LIN {X 0,Y 631.994,Z 1164.814,A -85,B 0,C 180,E1 28881.357,E2 28881.357} C_VEL
LIN {X 0,Y 632.102,Z 1158.024,A -85,B 0,C 180,E1 28878.874,E2 28878.874} C_VEL
LIN {X 0,Y 632.325,Z 1150.394,A -85,B 0,C 180,E1 28876.653,E2 28876.653} C_VEL
LIN {X 0,Y 632.601,Z 1142.497,A -85,B 0,C 180,E1 28874.696,E2 28874.696} C_VEL
LIN {X 0,Y 633.008,Z 1133.821,A -85,B 0,C 180,E1 28872.821,E2 28872.821} C_VEL
LIN {X 0,Y 633.525,Z 1124.191,A -85,B 0,C 180,E1 28870.98,E2 28870.98} C_VEL
LIN {X 0,Y 634.156,Z 1113.94,A -85,B 0,C 180,E1 28869.223,E2 28869.223} C_VEL
LIN {X 0,Y 635.003,Z 1101.645,A -85,B 0,C 180,E1 28867.329,E2 28867.329} C_VEL
LIN {X 0,Y 636.328,Z 1084.564,A -85,B 0,C 180,E1 28864.997,E2 28864.997} C_VEL
LIN {X 0,Y 637.814,Z 1067.276,A -85,B 0,C 180,E1 28862.93,E2 28862.93} C_VEL
LIN {X 0,Y 639.378,Z 1049.829,A -85,B 0,C 180,E1 28861.064,E2 28861.064} C_VEL
LIN {X 0,Y 641.404,Z 1029.08,A -85,B 0,C 180,E1 28859.094,E2 28859.094} C_VEL
LIN {X 0,Y 643.497,Z 1007.241,A -85,B 0,C 180,E1 28857.268,E2 28857.268} C_VEL
LIN {X 0,Y 645.579,Z 985.802,A -85,B 0,C 180,E1 28855.685,E2 28855.685} C_VEL
LIN {X 0,Y 647.811,Z 962.992,A -85,B 0,C 180,E1 28854.2,E2 28854.2} C_VEL
LIN {X 0,Y 650.063,Z 938.345,A -85,B 0,C 180,E1 28852.81,E2 28852.81} C_VEL
LIN {X 0,Y 651.914,Z 916.669,A -85,B 0,C 180,E1 28851.748,E2 28851.748} C_VEL
LIN {X 0,Y 653.565,Z 895.996,A -85,B 0,C 180,E1 28850.865,E2 28850.865} C_VEL
LIN {X 0,Y 655.03,Z 875.301,A -85,B 0,C 180,E1 28850.098,E2 28850.098} C_VEL
LIN {X 0,Y 656.479,Z 853.031,A -85,B 0,C 180,E1 28849.401,E2 28849.401} C_VEL
LIN {X 0,Y 658.004,Z 825.778,A -85,B 0,C 180,E1 28848.715,E2 28848.715} C_VEL
LIN {X 0,Y 659.041,Z 799.065,A -85,B 0,C 180,E1 28848.225,E2 28848.225} C_VEL
LIN {X 0,Y 660.569,Z 719.951,A -85,B 0,C 180,E1 28847.17,E2 28847.17} C_VEL
LIN {X 0,Y 664.422,Z 504.082,A -85,B 0,C 180,E1 28844.295,E2 28844.295} C_VEL
LIN {X 0,Y 666.835,Z 372.662,A -85,B 0,C 180,E1 28842.494,E2 28842.494} C_VEL
LIN {X 0,Y 658.444,Z 360.413,A -85,B 0,C 180,E1 28841.489,E2 28841.489} C_VEL
LIN {X 0,Y 654.623,Z 355.427,A -85,B 0,C 180,E1 28841.024,E2 28841.024} C_VEL
LIN {X 0,Y 651.502,Z 352.423,A -85,B 0,C 180,E1 28840.655,E2 28840.655} C_VEL
LIN {X 0,Y 645.168,Z 346.235,A -85,B 0,C 180,E1 28839.884,E2 28839.884} C_VEL
LIN {X 0,Y 643.333,Z 344.576,A -85,B 0,C 180,E1 28839.644,E2 28839.644} C_VEL
LIN {X 0,Y 641.516,Z 340.875,A -85,B 0,C 180,E1 28838.798,E2 28838.798} C_VEL
LIN {X 0,Y 639.282,Z 337.191,A -85,B 0,C 180,E1 28837.83,E2 28837.83} C_VEL
LIN {X 0,Y 638.533,Z 335.639,A -85,B 0,C 180,E1 28837.45,E2 28837.45} C_VEL
LIN {X 0,Y 636.307,Z 332.09,A -85,B 0,C 180,E1 28836.436,E2 28836.436} C_VEL
LIN {X 0,Y 635.627,Z 330.502,A -85,B 0,C 180,E1 28836.039,E2 28836.039} C_VEL
LIN {X 0,Y 633.306,Z 327.165,A -85,B 0,C 180,E1 28834.968,E2 28834.968} C_VEL
LIN {X 0,Y 632.884,Z 325.37,A -85,B 0,C 180,E1 28834.554,E2 28834.554} C_VEL
LIN {X 0,Y 632.898,Z 325.398,A -85,B 0,C 180,E1 28831.277,E2 28831.277} C_VEL
LIN {X 0,Y 632.862,Z 325.373,A -85,B 0,C 180,E1 28828.167,E2 28828.167} C_VEL
LIN {X 0,Y 632.883,Z 325.36,A -85,B 0,C 180,E1 28825.05,E2 28825.05} C_VEL
LIN {X 0,Y 632.867,Z 325.396,A -85,B 0,C 180,E1 28821.969,E2 28821.969} C_VEL
LIN {X 0,Y 632.884,Z 325.381,A -85,B 0,C 180,E1 28818.858,E2 28818.858} C_VEL
LIN {X 0,Y 632.886,Z 325.358,A -85,B 0,C 180,E1 28815.674,E2 28815.674} C_VEL
LIN {X 0,Y 632.89,Z 325.383,A -85,B 0,C 180,E1 28812.315,E2 28812.315} C_VEL
LIN {X 0,Y 632.866,Z 325.39,A -85,B 0,C 180,E1 28809.182,E2 28809.182} C_VEL
LIN {X 0,Y 632.874,Z 325.358,A -85,B 0,C 180,E1 28806.167,E2 28806.167} C_VEL
LIN {X 0,Y 632.873,Z 325.385,A -85,B 0,C 180,E1 28803.079,E2 28803.079} C_VEL
LIN {X 0,Y 632.863,Z 325.391,A -85,B 0,C 180,E1 28800,E2 28800} C_VEL
LIN {X 0,Y 632.888,Z 325.358,A -85,B 0,C 180,E1 28796.921,E2 28796.921} C_VEL
LIN {X 0,Y 632.914,Z 325.585,A -85,B 0,C 180,E1 28793.651,E2 28793.651} C_VEL
LIN {X 0,Y 634.17,Z 328.851,A -85,B 0,C 180,E1 28792.845,E2 28792.845} C_VEL
LIN {X 0,Y 636.114,Z 331.216,A -85,B 0,C 180,E1 28792.049,E2 28792.049} C_VEL
LIN {X 0,Y 637.819,Z 334.806,A -85,B 0,C 180,E1 28791.163,E2 28791.163} C_VEL
LIN {X 0,Y 639.201,Z 336.499,A -85,B 0,C 180,E1 28790.637,E2 28790.637} C_VEL
LIN {X 0,Y 641.051,Z 340.245,A -85,B 0,C 180,E1 28789.758,E2 28789.758} C_VEL
LIN {X 0,Y 642.203,Z 341.843,A -85,B 0,C 180,E1 28789.323,E2 28789.323} C_VEL
LIN {X 0,Y 644.496,Z 345.958,A -85,B 0,C 180,E1 28788.364,E2 28788.364} C_VEL
LIN {X 0,Y 647.578,Z 351.352,A -85,B 0,C 180,E1 28787.153,E2 28787.153} C_VEL
LIN {X 0,Y 653.401,Z 362.455,A -85,B 0,C 180,E1 28784.921,E2 28784.921} C_VEL
LIN {X 0,Y 659.977,Z 374.821,A -85,B 0,C 180,E1 28782.635,E2 28782.635} C_VEL
LIN {X 0,Y 666.865,Z 388.815,A -85,B 0,C 180,E1 28780.336,E2 28780.336} C_VEL
LIN {X 0,Y 664.135,Z 420.673,A -85,B 0,C 180,E1 28777.755,E2 28777.755} C_VEL
LIN {X 0,Y 661.315,Z 455.679,A -85,B 0,C 180,E1 28775.049,E2 28775.049} C_VEL
LIN {X 0,Y 658.271,Z 496.183,A -85,B 0,C 180,E1 28772.056,E2 28772.056} C_VEL
LIN {X 0,Y 655.36,Z 537.779,A -85,B 0,C 180,E1 28769.109,E2 28769.109} C_VEL
LIN {X 0,Y 654.216,Z 562.567,A -85,B 0,C 180,E1 28767.363,E2 28767.363} C_VEL
LIN {X 0,Y 655.292,Z 577.288,A -85,B 0,C 180,E1 28766.208,E2 28766.208} C_VEL
LIN {X 0,Y 657.897,Z 589.358,A -85,B 0,C 180,E1 28765.148,E2 28765.148} C_VEL
LIN {X 0,Y 662.309,Z 600.648,A -85,B 0,C 180,E1 28764.036,E2 28764.036} C_VEL
LIN {X 0,Y 668.439,Z 610.609,A -85,B 0,C 180,E1 28762.927,E2 28762.927} C_VEL
LIN {X 0,Y 676.331,Z 619.158,A -85,B 0,C 180,E1 28761.831,E2 28761.831} C_VEL
LIN {X 0,Y 685.342,Z 625.908,A -85,B 0,C 180,E1 28760.822,E2 28760.822} C_VEL
LIN {X 0,Y 695.344,Z 631.031,A -85,B 0,C 180,E1 28759.893,E2 28759.893} C_VEL
LIN {X 0,Y 700.807,Z 632.967,A -85,B 0,C 180,E1 28759.412,E2 28759.412} C_VEL
LIN {X 0,Y 704.135,Z 633.321,A -85,B 0,C 180,E1 28759,E2 28759} C_VEL
LIN {X 0,Y 706.593,Z 632.67,A -85,B 0,C 180,E1 28758.527,E2 28758.527} C_VEL
LIN {X 0,Y 707.801,Z 631.127,A -85,B 0,C 180,E1 28758.072,E2 28758.072} C_VEL
LIN {X 0,Y 707.787,Z 628.388,A -85,B 0,C 180,E1 28757.57,E2 28757.57} C_VEL
LIN {X 0,Y 706.223,Z 624.764,A -85,B 0,C 180,E1 28757.11,E2 28757.11} C_VEL
LIN {X 0,Y 703.206,Z 620.48,A -85,B 0,C 180,E1 28756.734,E2 28756.734} C_VEL
LIN {X 0,Y 694.622,Z 609.272,A -85,B 0,C 180,E1 28756.06,E2 28756.06} C_VEL
LIN {X 0,Y 687.011,Z 596.636,A -85,B 0,C 180,E1 28755.445,E2 28755.445} C_VEL
LIN {X 0,Y 682.904,Z 588.598,A -85,B 0,C 180,E1 28755.105,E2 28755.105} C_VEL
LIN {X 0,Y 678.866,Z 616.962,A -85,B 0,C 180,E1 28754.764,E2 28754.764} C_VEL
LIN {X 0,Y 675.836,Z 631.299,A -85,B 0,C 180,E1 28754.505,E2 28754.505} C_VEL
LIN {X 0,Y 673.585,Z 637.727,A -85,B 0,C 180,E1 28754.31,E2 28754.31} C_VEL
LIN {X 0,Y 669.429,Z 677.246,A -85,B 0,C 180,E1 28753.944,E2 28753.944} C_VEL
LIN {X 0,Y 665.551,Z 703.866,A -85,B 0,C 180,E1 28753.598,E2 28753.598} C_VEL
LIN {X 0,Y 662.995,Z 713.8,A -85,B 0,C 180,E1 28753.387,E2 28753.387} C_VEL
LIN {X 0,Y 661.297,Z 717.415,A -85,B 0,C 180,E1 28753.229,E2 28753.229} C_VEL
LIN {X 0,Y 659.009,Z 830.635,A -85,B 0,C 180,E1 28751.708,E2 28751.708} C_VEL
LIN {X 0,Y 657.873,Z 857.726,A -85,B 0,C 180,E1 28751.194,E2 28751.194} C_VEL
LIN {X 0,Y 656.431,Z 884.192,A -85,B 0,C 180,E1 28750.525,E2 28750.525} C_VEL
LIN {X 0,Y 654.785,Z 909.556,A -85,B 0,C 180,E1 28749.715,E2 28749.715} C_VEL
LIN {X 0,Y 652.732,Z 936.935,A -85,B 0,C 180,E1 28748.647,E2 28748.647} C_VEL
LIN {X 0,Y 650.615,Z 961.785,A -85,B 0,C 180,E1 28747.485,E2 28747.485} C_VEL
LIN {X 0,Y 648.417,Z 986.47,A -85,B 0,C 180,E1 28746.143,E2 28746.143} C_VEL
LIN {X 0,Y 646.162,Z 1010.12,A -85,B 0,C 180,E1 28744.656,E2 28744.656} C_VEL
LIN {X 0,Y 644.134,Z 1030.916,A -85,B 0,C 180,E1 28743.178,E2 28743.178} C_VEL
LIN {X 0,Y 641.929,Z 1053.565,A -85,B 0,C 180,E1 28741.347,E2 28741.347} C_VEL
LIN {X 0,Y 639.931,Z 1074.383,A -85,B 0,C 180,E1 28739.431,E2 28739.431} C_VEL
LIN {X 0,Y 638.122,Z 1093.746,A -85,B 0,C 180,E1 28737.429,E2 28737.429} C_VEL
LIN {X 0,Y 636.66,Z 1110.677,A -85,B 0,C 180,E1 28735.437,E2 28735.437} C_VEL
LIN {X 0,Y 635.437,Z 1125.874,A -85,B 0,C 180,E1 28733.454,E2 28733.454} C_VEL
LIN {X 0,Y 634.299,Z 1142.006,A -85,B 0,C 180,E1 28731.058,E2 28731.058} C_VEL
LIN {X 0,Y 633.468,Z 1155.309,A -85,B 0,C 180,E1 28728.782,E2 28728.782} C_VEL
LIN {X 0,Y 632.846,Z 1167.319,A -85,B 0,C 180,E1 28726.427,E2 28726.427} C_VEL
LIN {X 0,Y 632.418,Z 1177.763,A -85,B 0,C 180,E1 28723.997,E2 28723.997} C_VEL
LIN {X 0,Y 632.166,Z 1186.137,A -85,B 0,C 180,E1 28721.679,E2 28721.679} C_VEL
LIN {X 0,Y 632.007,Z 1193.403,A -85,B 0,C 180,E1 28719.167,E2 28719.167} C_VEL
LIN {X 0,Y 631.938,Z 1198.776,A -85,B 0,C 180,E1 28716.723,E2 28716.723} C_VEL
LIN {X 0,Y 631.918,Z 1202.393,A -85,B 0,C 180,E1 28714.355,E2 28714.355} C_VEL
LIN {X 0,Y 631.911,Z 1204.422,A -85,B 0,C 180,E1 28711.994,E2 28711.994} C_VEL
LIN {X 0,Y 631.892,Z 1204.916,A -85,B 0,C 180,E1 28709.546,E2 28709.546} C_VEL
LIN {X 0,Y 631.912,Z 1203.981,A -85,B 0,C 180,E1 28707.278,E2 28707.278} C_VEL
LIN {X 0,Y 631.925,Z 1201.414,A -85,B 0,C 180,E1 28704.915,E2 28704.915} C_VEL
LIN {X 0,Y 631.956,Z 1197.33,A -85,B 0,C 180,E1 28702.544,E2 28702.544} C_VEL
LIN {X 0,Y 632.039,Z 1191.654,A -85,B 0,C 180,E1 28700.161,E2 28700.161} C_VEL
LIN {X 0,Y 632.199,Z 1184.276,A -85,B 0,C 180,E1 28697.763,E2 28697.763} C_VEL
LIN {X 0,Y 632.542,Z 1174.752,A -85,B 0,C 180,E1 28695.255,E2 28695.255} C_VEL
LIN {X 0,Y 633.004,Z 1163.893,A -85,B 0,C 180,E1 28692.874,E2 28692.874} C_VEL
LIN {X 0,Y 633.621,Z 1152.683,A -85,B 0,C 180,E1 28690.742,E2 28690.742} C_VEL
LIN {X 0,Y 634.549,Z 1138.328,A -85,B 0,C 180,E1 28688.362,E2 28688.362} C_VEL
LIN {X 0,Y 635.659,Z 1122.981,A -85,B 0,C 180,E1 28686.154,E2 28686.154} C_VEL
LIN {X 0,Y 636.89,Z 1107.932,A -85,B 0,C 180,E1 28684.222,E2 28684.222} C_VEL
LIN {X 0,Y 638.608,Z 1088.547,A -85,B 0,C 180,E1 28682.016,E2 28682.016} C_VEL
LIN {X 0,Y 640.354,Z 1069.807,A -85,B 0,C 180,E1 28680.124,E2 28680.124} C_VEL
LIN {X 0,Y 642.484,Z 1047.697,A -85,B 0,C 180,E1 28678.157,E2 28678.157} C_VEL
LIN {X 0,Y 644.673,Z 1025.55,A -85,B 0,C 180,E1 28676.426,E2 28676.426} C_VEL
LIN {X 0,Y 646.945,Z 1001.819,A -85,B 0,C 180,E1 28674.795,E2 28674.795} C_VEL
LIN {X 0,Y 649.199,Z 977.864,A -85,B 0,C 180,E1 28673.364,E2 28673.364} C_VEL
LIN {X 0,Y 651.423,Z 953.129,A -85,B 0,C 180,E1 28672.088,E2 28672.088} C_VEL
LIN {X 0,Y 653.376,Z 928.962,A -85,B 0,C 180,E1 28671.025,E2 28671.025} C_VEL
LIN {X 0,Y 655.183,Z 903.445,A -85,B 0,C 180,E1 28670.078,E2 28670.078} C_VEL
LIN {X 0,Y 656.816,Z 877.86,A -85,B 0,C 180,E1 28669.299,E2 28669.299} C_VEL
LIN {X 0,Y 658.202,Z 851.179,A -85,B 0,C 180,E1 28668.662,E2 28668.662} C_VEL
LIN {X 0,Y 659.209,Z 824.645,A -85,B 0,C 180,E1 28668.201,E2 28668.201} C_VEL
LIN {X 0,Y 662.609,Z 643.494,A -85,B 0,C 180,E1 28665.792,E2 28665.792} C_VEL
LIN {X 0,Y 666.306,Z 614.925,A -85,B 0,C 180,E1 28665.248,E2 28665.248} C_VEL
LIN {X 0,Y 669.517,Z 589.966,A -85,B 0,C 180,E1 28664.86,E2 28664.86} C_VEL
LIN {X 0,Y 672.296,Z 566.613,A -85,B 0,C 180,E1 28664.405,E2 28664.405} C_VEL
LIN {X 0,Y 676.702,Z 531.964,A -85,B 0,C 180,E1 28663.91,E2 28663.91} C_VEL
LIN {X 0,Y 678.593,Z 513.611,A -85,B 0,C 180,E1 28663.531,E2 28663.531} C_VEL
LIN {X 0,Y 682.368,Z 483.277,A -85,B 0,C 180,E1 28663.109,E2 28663.109} C_VEL
LIN {X 0,Y 684.257,Z 468.994,A -85,B 0,C 180,E1 28662.937,E2 28662.937} C_VEL
LIN {X 0,Y 685.384,Z 454.57,A -85,B 0,C 180,E1 28662.615,E2 28662.615} C_VEL
LIN {X 0,Y 688.482,Z 428.06,A -85,B 0,C 180,E1 28662.237,E2 28662.237} C_VEL
LIN {X 0,Y 692.279,Z 400.87,A -85,B 0,C 180,E1 28661.95,E2 28661.95} C_VEL
LIN {X 0,Y 692.646,Z 391.557,A -85,B 0,C 180,E1 28661.72,E2 28661.72} C_VEL
LIN {X 0,Y 687.73,Z 389.873,A -85,B 0,C 180,E1 28661.195,E2 28661.195} C_VEL
LIN {X 0,Y 679.673,Z 385.544,A -85,B 0,C 180,E1 28660.366,E2 28660.366} C_VEL
LIN {X 0,Y 672.667,Z 379.562,A -85,B 0,C 180,E1 28659.565,E2 28659.565} C_VEL
LIN {X 0,Y 665.553,Z 371.898,A -85,B 0,C 180,E1 28658.681,E2 28658.681} C_VEL
LIN {X 0,Y 651.572,Z 351.934,A -85,B 0,C 180,E1 28656.707,E2 28656.707} C_VEL
LIN {X 0,Y 644.016,Z 341.599,A -85,B 0,C 180,E1 28655.58,E2 28655.58} C_VEL
LIN {X 0,Y 640.98,Z 337.137,A -85,B 0,C 180,E1 28655.102,E2 28655.102} C_VEL
LIN {X 0,Y 637.808,Z 333.354,A -85,B 0,C 180,E1 28654.618,E2 28654.618} C_VEL
LIN {X 0,Y 636.716,Z 331.263,A -85,B 0,C 180,E1 28654.426,E2 28654.426} C_VEL
LIN {X 0,Y 634.02,Z 328.611,A -85,B 0,C 180,E1 28654.019,E2 28654.019} C_VEL
LIN {X 0,Y 632.886,Z 325.399,A -85,B 0,C 180,E1 28653.761,E2 28653.761} C_VEL
LIN {X 0,Y 632.881,Z 325.349,A -85,B 0,C 180,E1 28650.565,E2 28650.565} C_VEL
LIN {X 0,Y 632.887,Z 325.378,A -85,B 0,C 180,E1 28647.371,E2 28647.371} C_VEL
LIN {X 0,Y 632.89,Z 325.36,A -85,B 0,C 180,E1 28644.055,E2 28644.055} C_VEL
LIN {X 0,Y 632.888,Z 325.385,A -85,B 0,C 180,E1 28640.92,E2 28640.92} C_VEL
LIN {X 0,Y 632.879,Z 325.389,A -85,B 0,C 180,E1 28637.695,E2 28637.695} C_VEL
LIN {X 0,Y 632.887,Z 325.4,A -85,B 0,C 180,E1 28634.549,E2 28634.549} C_VEL
LIN {X 0,Y 632.896,Z 325.508,A -85,B 0,C 180,E1 28633.038,E2 28633.038} C_VEL
LIN {X 0,Y 636.068,Z 337.173,A -85,B 0,C 180,E1 28632.552,E2 28632.552} C_VEL
LIN {X 0,Y 636.101,Z 412.444,A -85,B 0,C 180,E1 28629.957,E2 28629.957} C_VEL
LIN {X 0,Y 636.466,Z 489.624,A -85,B 0,C 180,E1 28627.175,E2 28627.175} C_VEL
LIN {X 0,Y 636.644,Z 555.776,A -85,B 0,C 180,E1 28624.711,E2 28624.711} C_VEL
LIN {X 0,Y 636.403,Z 631.985,A -85,B 0,C 180,E1 28621.801,E2 28621.801} C_VEL
LIN {X 0,Y 635.814,Z 713.116,A -85,B 0,C 180,E1 28618.648,E2 28618.648} C_VEL
LIN {X 0,Y 635.079,Z 790.594,A -85,B 0,C 180,E1 28615.575,E2 28615.575} C_VEL
LIN {X 0,Y 634.453,Z 844.266,A -85,B 0,C 180,E1 28613.439,E2 28613.439} C_VEL
LIN {X 0,Y 634.266,Z 848.016,A -85,B 0,C 180,E1 28613.329,E2 28613.329} C_VEL
LIN {X 0,Y 633.819,Z 961.824,A -85,B 0,C 180,E1 28611.994,E2 28611.994} C_VEL
LIN {X 0,Y 633.8,Z 974.114,A -85,B 0,C 180,E1 28611.732,E2 28611.732} C_VEL
LIN {X 0,Y 633.75,Z 985.462,A -85,B 0,C 180,E1 28611.38,E2 28611.38} C_VEL
LIN {X 0,Y 633.654,Z 996.602,A -85,B 0,C 180,E1 28610.921,E2 28610.921} C_VEL
LIN {X 0,Y 633.488,Z 1009.403,A -85,B 0,C 180,E1 28610.238,E2 28610.238} C_VEL
LIN {X 0,Y 633.311,Z 1020.589,A -85,B 0,C 180,E1 28609.447,E2 28609.447} C_VEL
LIN {X 0,Y 633.143,Z 1029.118,A -85,B 0,C 180,E1 28608.707,E2 28608.707} C_VEL
LIN {X 0,Y 632.977,Z 1037.028,A -85,B 0,C 180,E1 28607.872,E2 28607.872} C_VEL
LIN {X 0,Y 632.842,Z 1043.546,A -85,B 0,C 180,E1 28607.035,E2 28607.035} C_VEL
LIN {X 0,Y 632.717,Z 1049.448,A -85,B 0,C 180,E1 28606.101,E2 28606.101} C_VEL
LIN {X 0,Y 632.611,Z 1055.079,A -85,B 0,C 180,E1 28604.958,E2 28604.958} C_VEL
LIN {X 0,Y 632.522,Z 1059.484,A -85,B 0,C 180,E1 28603.648,E2 28603.648} C_VEL
LIN {X 0,Y 632.481,Z 1061.792,A -85,B 0,C 180,E1 28602.52,E2 28602.52} C_VEL
LIN {X 0,Y 632.459,Z 1062.804,A -85,B 0,C 180,E1 28601.472,E2 28601.472} C_VEL
LIN {X 0,Y 632.451,Z 1062.728,A -85,B 0,C 180,E1 28600.417,E2 28600.417} C_VEL
LIN {X 0,Y 632.453,Z 1061.4,A -85,B 0,C 180,E1 28599.259,E2 28599.259} C_VEL
LIN {X 0,Y 632.506,Z 1058.044,A -85,B 0,C 180,E1 28597.877,E2 28597.877} C_VEL
LIN {X 0,Y 632.565,Z 1053.404,A -85,B 0,C 180,E1 28596.691,E2 28596.691} C_VEL
LIN {X 0,Y 632.647,Z 1048.455,A -85,B 0,C 180,E1 28595.737,E2 28595.737} C_VEL
LIN {X 0,Y 632.771,Z 1041.957,A -85,B 0,C 180,E1 28594.745,E2 28594.745} C_VEL
LIN {X 0,Y 632.969,Z 1032.891,A -85,B 0,C 180,E1 28593.647,E2 28593.647} C_VEL
LIN {X 0,Y 633.021,Z 1029.911,A -85,B 0,C 180,E1 28593.355,E2 28593.355} C_VEL
LIN {X 0,Y 632.139,Z 1024.731,A -85,B 0,C 180,E1 28592.842,E2 28592.842} C_VEL
LIN {X 0,Y 627.932,Z 1014.736,A -85,B 0,C 180,E1 28591.965,E2 28591.965} C_VEL
LIN {X 0,Y 625.917,Z 1007.927,A -85,B 0,C 180,E1 28591.476,E2 28591.476} C_VEL
LIN {X 0,Y 625.646,Z 1004.089,A -85,B 0,C 180,E1 28591.253,E2 28591.253} C_VEL
LIN {X 0,Y 625.809,Z 992.507,A -85,B 0,C 180,E1 28590.678,E2 28590.678} C_VEL
LIN {X 0,Y 625.938,Z 977.574,A -85,B 0,C 180,E1 28590.131,E2 28590.131} C_VEL
LIN {X 0,Y 625.985,Z 964.18,A -85,B 0,C 180,E1 28589.811,E2 28589.811} C_VEL
LIN {X 0,Y 625.981,Z 947.83,A -85,B 0,C 180,E1 28589.577,E2 28589.577} C_VEL
LIN {X 0,Y 626.54,Z 844.713,A -85,B 0,C 180,E1 28588.355,E2 28588.355} C_VEL
LIN {X 0,Y 627.478,Z 776.547,A -85,B 0,C 180,E1 28585.577,E2 28585.577} C_VEL
LIN {X 0,Y 628.54,Z 696.106,A -85,B 0,C 180,E1 28582.287,E2 28582.287} C_VEL
LIN {X 0,Y 629.581,Z 616.689,A -85,B 0,C 180,E1 28579.04,E2 28579.04} C_VEL
LIN {X 0,Y 630.11,Z 578.008,A -85,B 0,C 180,E1 28577.445,E2 28577.445} C_VEL
LIN {X 0,Y 631.379,Z 580.022,A -85,B 0,C 180,E1 28577.296,E2 28577.296} C_VEL
LIN {X 0,Y 633.349,Z 580.034,A -85,B 0,C 180,E1 28577.122,E2 28577.122} C_VEL
LIN {X 0,Y 636.087,Z 577.689,A -85,B 0,C 180,E1 28576.921,E2 28576.921} C_VEL
LIN {X 0,Y 639.873,Z 571.769,A -85,B 0,C 180,E1 28576.686,E2 28576.686} C_VEL
LIN {X 0,Y 643.423,Z 570.526,A -85,B 0,C 180,E1 28576.405,E2 28576.405} C_VEL
LIN {X 0,Y 647.315,Z 567.094,A -85,B 0,C 180,E1 28576.133,E2 28576.133} C_VEL
LIN {X 0,Y 650.544,Z 562.61,A -85,B 0,C 180,E1 28575.933,E2 28575.933} C_VEL
LIN {X 0,Y 655.119,Z 559.939,A -85,B 0,C 180,E1 28575.589,E2 28575.589} C_VEL
LIN {X 0,Y 657.788,Z 557.468,A -85,B 0,C 180,E1 28575.39,E2 28575.39} C_VEL
LIN {X 0,Y 653.54,Z 783.546,A -85,B 0,C 180,E1 28572.379,E2 28572.379} C_VEL
LIN {X 0,Y 652.535,Z 812.346,A -85,B 0,C 180,E1 28571.928,E2 28571.928} C_VEL
LIN {X 0,Y 651.406,Z 835.088,A -85,B 0,C 180,E1 28571.443,E2 28571.443} C_VEL
LIN {X 0,Y 650.096,Z 856.645,A -85,B 0,C 180,E1 28570.867,E2 28570.867} C_VEL
LIN {X 0,Y 648.604,Z 878.002,A -85,B 0,C 180,E1 28570.178,E2 28570.178} C_VEL
LIN {X 0,Y 646.993,Z 899.085,A -85,B 0,C 180,E1 28569.376,E2 28569.376} C_VEL
LIN {X 0,Y 644.884,Z 923.987,A -85,B 0,C 180,E1 28568.275,E2 28568.275} C_VEL
LIN {X 0,Y 642.385,Z 949.606,A -85,B 0,C 180,E1 28566.929,E2 28566.929} C_VEL
LIN {X 0,Y 640.303,Z 970.247,A -85,B 0,C 180,E1 28565.686,E2 28565.686} C_VEL
LIN {X 0,Y 638.103,Z 991.626,A -85,B 0,C 180,E1 28564.233,E2 28564.233} C_VEL
LIN {X 0,Y 635.712,Z 1014.829,A -85,B 0,C 180,E1 28562.436,E2 28562.436} C_VEL
LIN {X 0,Y 633.494,Z 1035.642,A -85,B 0,C 180,E1 28560.6,E2 28560.6} C_VEL
LIN {X 0,Y 631.614,Z 1054.139,A -85,B 0,C 180,E1 28558.768,E2 28558.768} C_VEL
LIN {X 0,Y 629.755,Z 1073.595,A -85,B 0,C 180,E1 28556.6,E2 28556.6} C_VEL
LIN {X 0,Y 628.217,Z 1090.556,A -85,B 0,C 180,E1 28554.437,E2 28554.437} C_VEL
LIN {X 0,Y 627.143,Z 1103.497,A -85,B 0,C 180,E1 28552.597,E2 28552.597} C_VEL
LIN {X 0,Y 626.287,Z 1115.135,A -85,B 0,C 180,E1 28550.759,E2 28550.759} C_VEL
LIN {X 0,Y 625.562,Z 1126.046,A -85,B 0,C 180,E1 28548.838,E2 28548.838} C_VEL
LIN {X 0,Y 624.907,Z 1137.993,A -85,B 0,C 180,E1 28546.453,E2 28546.453} C_VEL
LIN {X 0,Y 624.452,Z 1147.909,A -85,B 0,C 180,E1 28544.087,E2 28544.087} C_VEL
LIN {X 0,Y 624.19,Z 1155.641,A -85,B 0,C 180,E1 28541.927,E2 28541.927} C_VEL
LIN {X 0,Y 624.038,Z 1162.223,A -85,B 0,C 180,E1 28539.687,E2 28539.687} C_VEL
LIN {X 0,Y 623.956,Z 1167.407,A -85,B 0,C 180,E1 28537.459,E2 28537.459} C_VEL
LIN {X 0,Y 623.925,Z 1171.503,A -85,B 0,C 180,E1 28535.058,E2 28535.058} C_VEL
LIN {X 0,Y 623.907,Z 1174.114,A -85,B 0,C 180,E1 28532.481,E2 28532.481} C_VEL
LIN {X 0,Y 623.908,Z 1174.944,A -85,B 0,C 180,E1 28530.093,E2 28530.093} C_VEL
LIN {X 0,Y 623.91,Z 1174.275,A -85,B 0,C 180,E1 28527.705,E2 28527.705} C_VEL
LIN {X 0,Y 623.913,Z 1172.101,A -85,B 0,C 180,E1 28525.313,E2 28525.313} C_VEL
LIN {X 0,Y 623.957,Z 1167.988,A -85,B 0,C 180,E1 28522.726,E2 28522.726} C_VEL
LIN {X 0,Y 624.032,Z 1162.716,A -85,B 0,C 180,E1 28520.409,E2 28520.409} C_VEL
LIN {X 0,Y 624.185,Z 1156.237,A -85,B 0,C 180,E1 28518.169,E2 28518.169} C_VEL
LIN {X 0,Y 624.414,Z 1148.973,A -85,B 0,C 180,E1 28516.103,E2 28516.103} C_VEL
LIN {X 0,Y 624.757,Z 1140.857,A -85,B 0,C 180,E1 28514.118,E2 28514.118} C_VEL
LIN {X 0,Y 625.336,Z 1130.094,A -85,B 0,C 180,E1 28511.834,E2 28511.834} C_VEL
LIN {X 0,Y 626.166,Z 1116.849,A -85,B 0,C 180,E1 28509.434,E2 28509.434} C_VEL
LIN {X 0,Y 627.043,Z 1104.749,A -85,B 0,C 180,E1 28507.5,E2 28507.5} C_VEL
LIN {X 0,Y 628.102,Z 1091.87,A -85,B 0,C 180,E1 28505.652,E2 28505.652} C_VEL
LIN {X 0,Y 629.351,Z 1077.487,A -85,B 0,C 180,E1 28503.791,E2 28503.791} C_VEL
LIN {X 0,Y 631.2,Z 1058.722,A -85,B 0,C 180,E1 28501.627,E2 28501.627} C_VEL
LIN {X 0,Y 633.129,Z 1039.206,A -85,B 0,C 180,E1 28499.646,E2 28499.646} C_VEL
LIN {X 0,Y 635.237,Z 1019.033,A -85,B 0,C 180,E1 28497.829,E2 28497.829} C_VEL
LIN {X 0,Y 637.525,Z 997.571,A -85,B 0,C 180,E1 28496.114,E2 28496.114} C_VEL
LIN {X 0,Y 639.937,Z 973.975,A -85,B 0,C 180,E1 28494.464,E2 28494.464} C_VEL
LIN {X 0,Y 642.052,Z 952.78,A -85,B 0,C 180,E1 28493.163,E2 28493.163} C_VEL
LIN {X 0,Y 644.106,Z 931.535,A -85,B 0,C 180,E1 28492.013,E2 28492.013} C_VEL
LIN {X 0,Y 646.501,Z 905.473,A -85,B 0,C 180,E1 28490.792,E2 28490.792} C_VEL
LIN {X 0,Y 648.49,Z 879.592,A -85,B 0,C 180,E1 28489.787,E2 28489.787} C_VEL
LIN {X 0,Y 650.03,Z 857.754,A -85,B 0,C 180,E1 28489.076,E2 28489.076} C_VEL
LIN {X 0,Y 651.348,Z 836.156,A -85,B 0,C 180,E1 28488.494,E2 28488.494} C_VEL
LIN {X 0,Y 652.45,Z 814.134,A -85,B 0,C 180,E1 28488.017,E2 28488.017} C_VEL
LIN {X 0,Y 653.358,Z 790.041,A -85,B 0,C 180,E1 28487.623,E2 28487.623} C_VEL
LIN {X 0,Y 657.651,Z 564.398,A -85,B 0,C 180,E1 28484.614,E2 28484.614} C_VEL
LIN {X 0,Y 661.429,Z 376.651,A -85,B 0,C 180,E1 28482.043,E2 28482.043} C_VEL
LIN {X 0,Y 652.563,Z 363.675,A -85,B 0,C 180,E1 28480.952,E2 28480.952} C_VEL
LIN {X 0,Y 648.863,Z 359.804,A -85,B 0,C 180,E1 28480.506,E2 28480.506} C_VEL
LIN {X 0,Y 640.93,Z 352.259,A -85,B 0,C 180,E1 28479.532,E2 28479.532} C_VEL
LIN {X 0,Y 637.437,Z 348.791,A -85,B 0,C 180,E1 28479.065,E2 28479.065} C_VEL
LIN {X 0,Y 636.389,Z 346.846,A -85,B 0,C 180,E1 28478.592,E2 28478.592} C_VEL
LIN {X 0,Y 634.261,Z 342.898,A -85,B 0,C 180,E1 28477.596,E2 28477.596} C_VEL
LIN {X 0,Y 631.483,Z 338.298,A -85,B 0,C 180,E1 28476.301,E2 28476.301} C_VEL
LIN {X 0,Y 630.765,Z 336.796,A -85,B 0,C 180,E1 28475.904,E2 28475.904} C_VEL
LIN {X 0,Y 628.536,Z 333.398,A -85,B 0,C 180,E1 28474.828,E2 28474.828} C_VEL
LIN {X 0,Y 628.008,Z 331.711,A -85,B 0,C 180,E1 28474.418,E2 28474.418} C_VEL
LIN {X 0,Y 625.558,Z 328.573,A -85,B 0,C 180,E1 28473.247,E2 28473.247} C_VEL
LIN {X 0,Y 624.923,Z 326.354,A -85,B 0,C 180,E1 28472.63,E2 28472.63} C_VEL
LIN {X 0,Y 624.954,Z 326.344,A -85,B 0,C 180,E1 28469.629,E2 28469.629} C_VEL
LIN {X 0,Y 624.948,Z 326.372,A -85,B 0,C 180,E1 28466.308,E2 28466.308} C_VEL
LIN {X 0,Y 624.961,Z 326.38,A -85,B 0,C 180,E1 28462.978,E2 28462.978} C_VEL
LIN {X 0,Y 624.923,Z 326.349,A -85,B 0,C 180,E1 28459.926,E2 28459.926} C_VEL
LIN {X 0,Y 624.945,Z 326.365,A -85,B 0,C 180,E1 28456.834,E2 28456.834} C_VEL
LIN {X 0,Y 624.932,Z 326.383,A -85,B 0,C 180,E1 28453.698,E2 28453.698} C_VEL
LIN {X 0,Y 624.942,Z 326.344,A -85,B 0,C 180,E1 28450.603,E2 28450.603} C_VEL
LIN {X 0,Y 624.951,Z 326.363,A -85,B 0,C 180,E1 28447.446,E2 28447.446} C_VEL
LIN {X 0,Y 624.951,Z 326.385,A -85,B 0,C 180,E1 28444.129,E2 28444.129} C_VEL
LIN {X 0,Y 624.922,Z 326.351,A -85,B 0,C 180,E1 28441.008,E2 28441.008} C_VEL
LIN {X 0,Y 624.936,Z 326.351,A -85,B 0,C 180,E1 28437.983,E2 28437.983} C_VEL
LIN {X 0,Y 624.948,Z 326.484,A -85,B 0,C 180,E1 28435.549,E2 28435.549} C_VEL
LIN {X 0,Y 626.13,Z 329.671,A -85,B 0,C 180,E1 28434.685,E2 28434.685} C_VEL
LIN {X 0,Y 628.21,Z 331.939,A -85,B 0,C 180,E1 28433.787,E2 28433.787} C_VEL
LIN {X 0,Y 629.658,Z 335.462,A -85,B 0,C 180,E1 28432.885,E2 28432.885} C_VEL
LIN {X 0,Y 631.371,Z 337.57,A -85,B 0,C 180,E1 28432.172,E2 28432.172} C_VEL
LIN {X 0,Y 633.296,Z 341.416,A -85,B 0,C 180,E1 28431.19,E2 28431.19} C_VEL
LIN {X 0,Y 634.425,Z 342.855,A -85,B 0,C 180,E1 28430.749,E2 28430.749} C_VEL
LIN {X 0,Y 636.517,Z 346.864,A -85,B 0,C 180,E1 28429.775,E2 28429.775} C_VEL
LIN {X 0,Y 637.56,Z 348.635,A -85,B 0,C 180,E1 28429.335,E2 28429.335} C_VEL
LIN {X 0,Y 640.285,Z 353.504,A -85,B 0,C 180,E1 28428.195,E2 28428.195} C_VEL
LIN {X 0,Y 643.723,Z 359.924,A -85,B 0,C 180,E1 28426.801,E2 28426.801} C_VEL
LIN {X 0,Y 648.092,Z 367.88,A -85,B 0,C 180,E1 28425.161,E2 28425.161} C_VEL
LIN {X 0,Y 654.802,Z 380.744,A -85,B 0,C 180,E1 28422.768,E2 28422.768} C_VEL
LIN {X 0,Y 661.155,Z 393.692,A -85,B 0,C 180,E1 28420.612,E2 28420.612} C_VEL
LIN {X 0,Y 658.22,Z 425.64,A -85,B 0,C 180,E1 28418.009,E2 28418.009} C_VEL
LIN {X 0,Y 655.209,Z 460.692,A -85,B 0,C 180,E1 28415.283,E2 28415.283} C_VEL
LIN {X 0,Y 651.826,Z 502.805,A -85,B 0,C 180,E1 28412.154,E2 28412.154} C_VEL
LIN {X 0,Y 648.792,Z 543.372,A -85,B 0,C 180,E1 28409.263,E2 28409.263} C_VEL
LIN {X 0,Y 647.736,Z 565.785,A -85,B 0,C 180,E1 28407.664,E2 28407.664} C_VEL
LIN {X 0,Y 648.737,Z 580.584,A -85,B 0,C 180,E1 28406.491,E2 28406.491} C_VEL
LIN {X 0,Y 651.413,Z 593.402,A -85,B 0,C 180,E1 28405.356,E2 28405.356} C_VEL
LIN {X 0,Y 655.925,Z 605.161,A -85,B 0,C 180,E1 28404.189,E2 28404.189} C_VEL
LIN {X 0,Y 662.053,Z 615.326,A -85,B 0,C 180,E1 28403.051,E2 28403.051} C_VEL
LIN {X 0,Y 669.834,Z 624.044,A -85,B 0,C 180,E1 28401.939,E2 28401.939} C_VEL
LIN {X 0,Y 678.71,Z 631.028,A -85,B 0,C 180,E1 28400.91,E2 28400.91} C_VEL
LIN {X 0,Y 688.549,Z 636.454,A -85,B 0,C 180,E1 28399.961,E2 28399.961} C_VEL
LIN {X 0,Y 697.023,Z 639.68,A -85,B 0,C 180,E1 28399.235,E2 28399.235} C_VEL
LIN {X 0,Y 700.911,Z 640.124,A -85,B 0,C 180,E1 28398.771,E2 28398.771} C_VEL
LIN {X 0,Y 703.576,Z 639.334,A -85,B 0,C 180,E1 28398.252,E2 28398.252} C_VEL
LIN {X 0,Y 704.754,Z 637.446,A -85,B 0,C 180,E1 28397.739,E2 28397.739} C_VEL
LIN {X 0,Y 704.453,Z 634.48,A -85,B 0,C 180,E1 28397.235,E2 28397.235} C_VEL
LIN {X 0,Y 702.644,Z 630.811,A -85,B 0,C 180,E1 28396.795,E2 28396.795} C_VEL
LIN {X 0,Y 699.406,Z 626.509,A -85,B 0,C 180,E1 28396.437,E2 28396.437} C_VEL
LIN {X 0,Y 690.583,Z 614.969,A -85,B 0,C 180,E1 28395.736,E2 28395.736} C_VEL
LIN {X 0,Y 686.077,Z 608.132,A -85,B 0,C 180,E1 28395.368,E2 28395.368} C_VEL
LIN {X 0,Y 682.44,Z 628.725,A -85,B 0,C 180,E1 28395.066,E2 28395.066} C_VEL
LIN {X 0,Y 679.702,Z 638.436,A -85,B 0,C 180,E1 28394.835,E2 28394.835} C_VEL
LIN {X 0,Y 678.954,Z 640.925,A -85,B 0,C 180,E1 28394.772,E2 28394.772} C_VEL
LIN {X 0,Y 674.72,Z 680.224,A -85,B 0,C 180,E1 28394.408,E2 28394.408} C_VEL
LIN {X 0,Y 671.52,Z 698.99,A -85,B 0,C 180,E1 28394.221,E2 28394.221} C_VEL
LIN {X 0,Y 667.827,Z 712.519,A -85,B 0,C 180,E1 28394.056,E2 28394.056} C_VEL
LIN {X 0,Y 664.966,Z 720.078,A -85,B 0,C 180,E1 28393.851,E2 28393.851} C_VEL
LIN {X 0,Y 664.204,Z 722.06,A -85,B 0,C 180,E1 28393.796,E2 28393.796} C_VEL
LIN {X 0,Y 660.337,Z 733.945,A -85,B 0,C 180,E1 28393.696,E2 28393.696} C_VEL
LIN {X 0,Y 656.716,Z 743.078,A -85,B 0,C 180,E1 28393.485,E2 28393.485} C_VEL
LIN {X 0,Y 654.734,Z 748.123,A -85,B 0,C 180,E1 28393.286,E2 28393.286} C_VEL
LIN {X 0,Y 653.055,Z 829.87,A -85,B 0,C 180,E1 28392.188,E2 28392.188} C_VEL
LIN {X 0,Y 651.857,Z 857.189,A -85,B 0,C 180,E1 28391.673,E2 28391.673} C_VEL
LIN {X 0,Y 650.353,Z 883.418,A -85,B 0,C 180,E1 28391.011,E2 28391.011} C_VEL
LIN {X 0,Y 648.596,Z 908.685,A -85,B 0,C 180,E1 28390.205,E2 28390.205} C_VEL
LIN {X 0,Y 646.599,Z 934.08,A -85,B 0,C 180,E1 28389.218,E2 28389.218} C_VEL
LIN {X 0,Y 644.381,Z 958.786,A -85,B 0,C 180,E1 28388.081,E2 28388.081} C_VEL
LIN {X 0,Y 642.058,Z 983.073,A -85,B 0,C 180,E1 28386.781,E2 28386.781} C_VEL
LIN {X 0,Y 639.563,Z 1007.939,A -85,B 0,C 180,E1 28385.23,E2 28385.23} C_VEL
LIN {X 0,Y 637.37,Z 1029.001,A -85,B 0,C 180,E1 28383.733,E2 28383.733} C_VEL
LIN {X 0,Y 635.125,Z 1050.057,A -85,B 0,C 180,E1 28382.04,E2 28382.04} C_VEL
LIN {X 0,Y 632.904,Z 1071.52,A -85,B 0,C 180,E1 28380.088,E2 28380.088} C_VEL
LIN {X 0,Y 631.121,Z 1089.387,A -85,B 0,C 180,E1 28378.251,E2 28378.251} C_VEL
LIN {X 0,Y 629.253,Z 1108.732,A -85,B 0,C 180,E1 28376.011,E2 28376.011} C_VEL
LIN {X 0,Y 627.947,Z 1123.71,A -85,B 0,C 180,E1 28374.055,E2 28374.055} C_VEL
LIN {X 0,Y 626.699,Z 1139.553,A -85,B 0,C 180,E1 28371.723,E2 28371.723} C_VEL
LIN {X 0,Y 625.753,Z 1153.221,A -85,B 0,C 180,E1 28369.411,E2 28369.411} C_VEL
LIN {X 0,Y 625.091,Z 1164.323,A -85,B 0,C 180,E1 28367.261,E2 28367.261} C_VEL
LIN {X 0,Y 624.601,Z 1174.76,A -85,B 0,C 180,E1 28364.934,E2 28364.934} C_VEL
LIN {X 0,Y 624.235,Z 1184.285,A -85,B 0,C 180,E1 28362.393,E2 28362.393} C_VEL
LIN {X 0,Y 624.054,Z 1191.66,A -85,B 0,C 180,E1 28359.963,E2 28359.963} C_VEL
LIN {X 0,Y 623.958,Z 1197.334,A -85,B 0,C 180,E1 28357.55,E2 28357.55} C_VEL
LIN {X 0,Y 623.925,Z 1201.417,A -85,B 0,C 180,E1 28355.148,E2 28355.148} C_VEL
LIN {X 0,Y 623.912,Z 1203.982,A -85,B 0,C 180,E1 28352.755,E2 28352.755} C_VEL
LIN {X 0,Y 623.892,Z 1204.916,A -85,B 0,C 180,E1 28350.458,E2 28350.458} C_VEL
LIN {X 0,Y 623.911,Z 1204.419,A -85,B 0,C 180,E1 28347.978,E2 28347.978} C_VEL
LIN {X 0,Y 623.917,Z 1202.391,A -85,B 0,C 180,E1 28345.587,E2 28345.587} C_VEL
LIN {X 0,Y 623.94,Z 1198.772,A -85,B 0,C 180,E1 28343.188,E2 28343.188} C_VEL
LIN {X 0,Y 624.016,Z 1193.539,A -85,B 0,C 180,E1 28340.77,E2 28340.77} C_VEL
LIN {X 0,Y 624.181,Z 1186.435,A -85,B 0,C 180,E1 28338.261,E2 28338.261} C_VEL
LIN {X 0,Y 624.441,Z 1178.472,A -85,B 0,C 180,E1 28336.007,E2 28336.007} C_VEL
LIN {X 0,Y 624.875,Z 1168.591,A -85,B 0,C 180,E1 28333.642,E2 28333.642} C_VEL
LIN {X 0,Y 625.568,Z 1156.145,A -85,B 0,C 180,E1 28331.128,E2 28331.128} C_VEL
LIN {X 0,Y 626.44,Z 1143.14,A -85,B 0,C 180,E1 28328.854,E2 28328.854} C_VEL
LIN {X 0,Y 627.605,Z 1127.93,A -85,B 0,C 180,E1 28326.528,E2 28326.528} C_VEL
LIN {X 0,Y 629.024,Z 1111.437,A -85,B 0,C 180,E1 28324.33,E2 28324.33} C_VEL
LIN {X 0,Y 630.586,Z 1094.58,A -85,B 0,C 180,E1 28322.315,E2 28322.315} C_VEL
LIN {X 0,Y 632.575,Z 1074.853,A -85,B 0,C 180,E1 28320.242,E2 28320.242} C_VEL
LIN {X 0,Y 634.665,Z 1054.695,A -85,B 0,C 180,E1 28318.356,E2 28318.356} C_VEL
LIN {X 0,Y 637.117,Z 1031.366,A -85,B 0,C 180,E1 28316.445,E2 28316.445} C_VEL
LIN {X 0,Y 639.332,Z 1010.088,A -85,B 0,C 180,E1 28314.917,E2 28314.917} C_VEL
LIN {X 0,Y 641.735,Z 986.425,A -85,B 0,C 180,E1 28313.417,E2 28313.417} C_VEL
LIN {X 0,Y 644.12,Z 961.497,A -85,B 0,C 180,E1 28312.054,E2 28312.054} C_VEL
LIN {X 0,Y 646.323,Z 937.364,A -85,B 0,C 180,E1 28310.918,E2 28310.918} C_VEL
LIN {X 0,Y 648.506,Z 910.081,A -85,B 0,C 180,E1 28309.843,E2 28309.843} C_VEL
LIN {X 0,Y 650.304,Z 884.072,A -85,B 0,C 180,E1 28309.008,E2 28309.008} C_VEL
LIN {X 0,Y 651.829,Z 857.661,A -85,B 0,C 180,E1 28308.338,E2 28308.338} C_VEL
LIN {X 0,Y 653.039,Z 830.34,A -85,B 0,C 180,E1 28307.819,E2 28307.819} C_VEL
LIN {X 0,Y 654.514,Z 759.757,A -85,B 0,C 180,E1 28306.867,E2 28306.867} C_VEL
LIN {X 0,Y 655.981,Z 690.855,A -85,B 0,C 180,E1 28305.937,E2 28305.937} C_VEL
LIN {X 0,Y 659.967,Z 656.067,A -85,B 0,C 180,E1 28305.302,E2 28305.302} C_VEL
LIN {X 0,Y 661.551,Z 641.994,A -85,B 0,C 180,E1 28305.056,E2 28305.056} C_VEL
LIN {X 0,Y 664.876,Z 611.059,A -85,B 0,C 180,E1 28304.51,E2 28304.51} C_VEL
LIN {X 0,Y 667.17,Z 591.276,A -85,B 0,C 180,E1 28304.212,E2 28304.212} C_VEL
LIN {X 0,Y 669.415,Z 567.124,A -85,B 0,C 180,E1 28303.767,E2 28303.767} C_VEL
LIN {X 0,Y 673.407,Z 533.187,A -85,B 0,C 180,E1 28303.298,E2 28303.298} C_VEL
LIN {X 0,Y 674.83,Z 513.773,A -85,B 0,C 180,E1 28302.929,E2 28302.929} C_VEL
LIN {X 0,Y 678.435,Z 482.816,A -85,B 0,C 180,E1 28302.519,E2 28302.519} C_VEL
LIN {X 0,Y 680.055,Z 470.137,A -85,B 0,C 180,E1 28302.368,E2 28302.368} C_VEL
LIN {X 0,Y 680.764,Z 454.491,A -85,B 0,C 180,E1 28302.061,E2 28302.061} C_VEL
LIN {X 0,Y 683.73,Z 427.188,A -85,B 0,C 180,E1 28301.697,E2 28301.697} C_VEL
LIN {X 0,Y 687.282,Z 401.897,A -85,B 0,C 180,E1 28301.43,E2 28301.43} C_VEL
LIN {X 0,Y 687.234,Z 398.213,A -85,B 0,C 180,E1 28301.342,E2 28301.342} C_VEL
LIN {X 0,Y 678.612,Z 394.106,A -85,B 0,C 180,E1 28300.47,E2 28300.47} C_VEL
LIN {X 0,Y 671.055,Z 388.359,A -85,B 0,C 180,E1 28299.623,E2 28299.623} C_VEL
LIN {X 0,Y 662.074,Z 378.905,A -85,B 0,C 180,E1 28298.506,E2 28298.506} C_VEL
LIN {X 0,Y 647.386,Z 357.913,A -85,B 0,C 180,E1 28296.404,E2 28296.404} C_VEL
LIN {X 0,Y 640.015,Z 347.804,A -85,B 0,C 180,E1 28295.286,E2 28295.286} C_VEL
LIN {X 0,Y 636.279,Z 342.714,A -85,B 0,C 180,E1 28294.699,E2 28294.699} C_VEL
LIN {X 0,Y 633.251,Z 338.253,A -85,B 0,C 180,E1 28294.203,E2 28294.203} C_VEL
LIN {X 0,Y 630.127,Z 334.712,A -85,B 0,C 180,E1 28293.71,E2 28293.71} C_VEL
LIN {X 0,Y 628.896,Z 332.335,A -85,B 0,C 180,E1 28293.484,E2 28293.484} C_VEL
LIN {X 0,Y 626.243,Z 329.882,A -85,B 0,C 180,E1 28293.07,E2 28293.07} C_VEL
LIN {X 0,Y 624.986,Z 326.767,A -85,B 0,C 180,E1 28292.811,E2 28292.811} C_VEL
LIN {X 0,Y 624.925,Z 326.348,A -85,B 0,C 180,E1 28292.767,E2 28292.767} C_VEL
LIN {X 0,Y 624.931,Z 326.362,A -85,B 0,C 180,E1 28289.68,E2 28289.68} C_VEL
LIN {X 0,Y 624.925,Z 326.341,A -85,B 0,C 180,E1 28286.718,E2 28286.718} C_VEL
LIN {X 0,Y 624.948,Z 326.369,A -85,B 0,C 180,E1 28283.478,E2 28283.478} C_VEL
LIN {X 0,Y 624.946,Z 326.372,A -85,B 0,C 180,E1 28280.316,E2 28280.316} C_VEL
LIN {X 0,Y 624.947,Z 326.371,A -85,B 0,C 180,E1 28277.025,E2 28277.025} C_VEL
LIN {X 0,Y 624.956,Z 326.386,A -85,B 0,C 180,E1 28273.792,E2 28273.792} C_VEL
LIN {X 0,Y 624.965,Z 326.482,A -85,B 0,C 180,E1 28273.243,E2 28273.243} C_VEL
LIN {X 0,Y 628.416,Z 339.108,A -85,B 0,C 180,E1 28272.712,E2 28272.712} C_VEL
LIN {X 0,Y 628.45,Z 420.666,A -85,B 0,C 180,E1 28269.894,E2 28269.894} C_VEL
LIN {X 0,Y 628.878,Z 502.02,A -85,B 0,C 180,E1 28266.94,E2 28266.94} C_VEL
LIN {X 0,Y 628.93,Z 575.151,A -85,B 0,C 180,E1 28264.194,E2 28264.194} C_VEL
LIN {X 0,Y 628.538,Z 653.354,A -85,B 0,C 180,E1 28261.185,E2 28261.185} C_VEL
LIN {X 0,Y 627.953,Z 726.616,A -85,B 0,C 180,E1 28258.312,E2 28258.312} C_VEL
LIN {X 0,Y 627.191,Z 803.813,A -85,B 0,C 180,E1 28255.245,E2 28255.245} C_VEL
LIN {X 0,Y 626.552,Z 846.459,A -85,B 0,C 180,E1 28253.54,E2 28253.54} C_VEL
LIN {X 0,Y 626.429,Z 849.807,A -85,B 0,C 180,E1 28253.458,E2 28253.458} C_VEL
LIN {X 0,Y 625.96,Z 963.074,A -85,B 0,C 180,E1 28252.11,E2 28252.11} C_VEL
LIN {X 0,Y 625.946,Z 975.457,A -85,B 0,C 180,E1 28251.841,E2 28251.841} C_VEL
LIN {X 0,Y 625.902,Z 986.29,A -85,B 0,C 180,E1 28251.502,E2 28251.502} C_VEL
LIN {X 0,Y 625.805,Z 997.514,A -85,B 0,C 180,E1 28251.038,E2 28251.038} C_VEL
LIN {X 0,Y 625.644,Z 1009.735,A -85,B 0,C 180,E1 28250.386,E2 28250.386} C_VEL
LIN {X 0,Y 625.453,Z 1021.634,A -85,B 0,C 180,E1 28249.546,E2 28249.546} C_VEL
LIN {X 0,Y 625.265,Z 1030.669,A -85,B 0,C 180,E1 28248.75,E2 28248.75} C_VEL
LIN {X 0,Y 625.093,Z 1038.525,A -85,B 0,C 180,E1 28247.904,E2 28247.904} C_VEL
LIN {X 0,Y 624.938,Z 1045.65,A -85,B 0,C 180,E1 28246.962,E2 28246.962} C_VEL
LIN {X 0,Y 624.776,Z 1052.913,A -85,B 0,C 180,E1 28245.732,E2 28245.732} C_VEL
LIN {X 0,Y 624.662,Z 1058.067,A -85,B 0,C 180,E1 28244.495,E2 28244.495} C_VEL
LIN {X 0,Y 624.595,Z 1061.16,A -85,B 0,C 180,E1 28243.444,E2 28243.444} C_VEL
LIN {X 0,Y 624.561,Z 1063.115,A -85,B 0,C 180,E1 28242.387,E2 28242.387} C_VEL
LIN {X 0,Y 624.532,Z 1064.012,A -85,B 0,C 180,E1 28241.228,E2 28241.228} C_VEL
LIN {X 0,Y 624.538,Z 1063.443,A -85,B 0,C 180,E1 28239.866,E2 28239.866} C_VEL
LIN {X 0,Y 624.551,Z 1061.144,A -85,B 0,C 180,E1 28238.591,E2 28238.591} C_VEL
LIN {X 0,Y 624.599,Z 1057.818,A -85,B 0,C 180,E1 28237.473,E2 28237.473} C_VEL
LIN {X 0,Y 624.667,Z 1053.388,A -85,B 0,C 180,E1 28236.411,E2 28236.411} C_VEL
LIN {X 0,Y 624.813,Z 1046.752,A -85,B 0,C 180,E1 28235.211,E2 28235.211} C_VEL
LIN {X 0,Y 624.981,Z 1038.551,A -85,B 0,C 180,E1 28234.102,E2 28234.102} C_VEL
LIN {X 0,Y 625.158,Z 1030.087,A -85,B 0,C 180,E1 28233.187,E2 28233.187} C_VEL
LIN {X 0,Y 625.35,Z 1020.862,A -85,B 0,C 180,E1 28232.374,E2 28232.374} C_VEL
LIN {X 0,Y 625.568,Z 1008.604,A -85,B 0,C 180,E1 28231.508,E2 28231.508} C_VEL
LIN {X 0,Y 625.646,Z 1004.089,A -85,B 0,C 180,E1 28231.253,E2 28231.253} C_VEL
LIN {X 0,Y 624.864,Z 997.495,A -85,B 0,C 180,E1 28230.886,E2 28230.886} C_VEL
LIN {X 0,Y 621.411,Z 987.108,A -85,B 0,C 180,E1 28230.365,E2 28230.365} C_VEL
LIN {X 0,Y 618.719,Z 978.22,A -85,B 0,C 180,E1 28230.012,E2 28230.012} C_VEL
LIN {X 0,Y 618.105,Z 972.983,A -85,B 0,C 180,E1 28229.858,E2 28229.858} C_VEL
LIN {X 0,Y 618.137,Z 957.176,A -85,B 0,C 180,E1 28229.548,E2 28229.548} C_VEL
LIN {X 0,Y 618.721,Z 845.652,A -85,B 0,C 180,E1 28228.208,E2 28228.208} C_VEL
LIN {X 0,Y 619.683,Z 781.766,A -85,B 0,C 180,E1 28225.587,E2 28225.587} C_VEL
LIN {X 0,Y 620.805,Z 700.963,A -85,B 0,C 180,E1 28222.263,E2 28222.263} C_VEL
LIN {X 0,Y 621.881,Z 622.711,A -85,B 0,C 180,E1 28219.047,E2 28219.047} C_VEL
LIN {X 0,Y 622.271,Z 594.249,A -85,B 0,C 180,E1 28217.867,E2 28217.867} C_VEL
LIN {X 0,Y 623.475,Z 596.288,A -85,B 0,C 180,E1 28217.719,E2 28217.719} C_VEL
LIN {X 0,Y 625.234,Z 596.423,A -85,B 0,C 180,E1 28217.555,E2 28217.555} C_VEL
LIN {X 0,Y 627.966,Z 594.371,A -85,B 0,C 180,E1 28217.35,E2 28217.35} C_VEL
LIN {X 0,Y 631.549,Z 588.961,A -85,B 0,C 180,E1 28217.125,E2 28217.125} C_VEL
LIN {X 0,Y 631.964,Z 588.18,A -85,B 0,C 180,E1 28217.102,E2 28217.102} C_VEL
LIN {X 0,Y 635.527,Z 586.99,A -85,B 0,C 180,E1 28216.812,E2 28216.812} C_VEL
LIN {X 0,Y 639.262,Z 583.74,A -85,B 0,C 180,E1 28216.544,E2 28216.544} C_VEL
LIN {X 0,Y 642.832,Z 578.909,A -85,B 0,C 180,E1 28216.321,E2 28216.321} C_VEL
LIN {X 0,Y 647.484,Z 576.142,A -85,B 0,C 180,E1 28215.979,E2 28215.979} C_VEL
LIN {X 0,Y 651.821,Z 571.879,A -85,B 0,C 180,E1 28215.692,E2 28215.692} C_VEL
LIN {X 0,Y 647.386,Z 791.63,A -85,B 0,C 180,E1 28212.742,E2 28212.742} C_VEL
LIN {X 0,Y 646.468,Z 814.431,A -85,B 0,C 180,E1 28212.364,E2 28212.364} C_VEL
LIN {X 0,Y 645.322,Z 835.987,A -85,B 0,C 180,E1 28211.895,E2 28211.895} C_VEL
LIN {X 0,Y 643.96,Z 857.072,A -85,B 0,C 180,E1 28211.327,E2 28211.327} C_VEL
LIN {X 0,Y 642.41,Z 878.014,A -85,B 0,C 180,E1 28210.646,E2 28210.646} C_VEL
LIN {X 0,Y 640.691,Z 899.112,A -85,B 0,C 180,E1 28209.84,E2 28209.84} C_VEL
LIN {X 0,Y 638.453,Z 923.995,A -85,B 0,C 180,E1 28208.732,E2 28208.732} C_VEL
LIN {X 0,Y 635.924,Z 948.578,A -85,B 0,C 180,E1 28207.436,E2 28207.436} C_VEL
LIN {X 0,Y 633.661,Z 969.55,A -85,B 0,C 180,E1 28206.169,E2 28206.169} C_VEL
LIN {X 0,Y 631.367,Z 990.221,A -85,B 0,C 180,E1 28204.76,E2 28204.76} C_VEL
LIN {X 0,Y 628.858,Z 1013.029,A -85,B 0,C 180,E1 28202.997,E2 28202.997} C_VEL
LIN {X 0,Y 626.477,Z 1034.064,A -85,B 0,C 180,E1 28201.14,E2 28201.14} C_VEL
LIN {X 0,Y 624.405,Z 1052.667,A -85,B 0,C 180,E1 28199.294,E2 28199.294} C_VEL
LIN {X 0,Y 622.599,Z 1070.2,A -85,B 0,C 180,E1 28197.344,E2 28197.344} C_VEL
LIN {X 0,Y 620.717,Z 1089.057,A -85,B 0,C 180,E1 28194.965,E2 28194.965} C_VEL
LIN {X 0,Y 619.494,Z 1102.852,A -85,B 0,C 180,E1 28192.993,E2 28192.993} C_VEL
LIN {X 0,Y 618.539,Z 1114.555,A -85,B 0,C 180,E1 28191.131,E2 28191.131} C_VEL
LIN {X 0,Y 617.795,Z 1125.006,A -85,B 0,C 180,E1 28189.28,E2 28189.28} C_VEL
LIN {X 0,Y 617.177,Z 1134.763,A -85,B 0,C 180,E1 28187.344,E2 28187.344} C_VEL
LIN {X 0,Y 616.657,Z 1144.95,A -85,B 0,C 180,E1 28185.037,E2 28185.037} C_VEL
LIN {X 0,Y 616.248,Z 1154.74,A -85,B 0,C 180,E1 28182.368,E2 28182.368} C_VEL
LIN {X 0,Y 616.074,Z 1161.478,A -85,B 0,C 180,E1 28180.096,E2 28180.096} C_VEL
LIN {X 0,Y 615.977,Z 1166.818,A -85,B 0,C 180,E1 28177.838,E2 28177.838} C_VEL
LIN {X 0,Y 615.928,Z 1170.807,A -85,B 0,C 180,E1 28175.591,E2 28175.591} C_VEL
LIN {X 0,Y 615.913,Z 1173.641,A -85,B 0,C 180,E1 28173.165,E2 28173.165} C_VEL
LIN {X 0,Y 615.894,Z 1174.888,A -85,B 0,C 180,E1 28170.652,E2 28170.652} C_VEL
LIN {X 0,Y 615.911,Z 1174.564,A -85,B 0,C 180,E1 28168.234,E2 28168.234} C_VEL
LIN {X 0,Y 615.918,Z 1172.896,A -85,B 0,C 180,E1 28165.998,E2 28165.998} C_VEL
LIN {X 0,Y 615.941,Z 1169.924,A -85,B 0,C 180,E1 28163.757,E2 28163.757} C_VEL
LIN {X 0,Y 615.997,Z 1165.633,A -85,B 0,C 180,E1 28161.507,E2 28161.507} C_VEL
LIN {X 0,Y 616.113,Z 1159.161,A -85,B 0,C 180,E1 28158.961,E2 28158.961} C_VEL
LIN {X 0,Y 616.374,Z 1151.446,A -85,B 0,C 180,E1 28156.588,E2 28156.588} C_VEL
LIN {X 0,Y 616.705,Z 1143.304,A -85,B 0,C 180,E1 28154.485,E2 28154.485} C_VEL
LIN {X 0,Y 617.207,Z 1134.277,A -85,B 0,C 180,E1 28152.464,E2 28152.464} C_VEL
LIN {X 0,Y 617.798,Z 1124.969,A -85,B 0,C 180,E1 28150.624,E2 28150.624} C_VEL
LIN {X 0,Y 618.537,Z 1114.515,A -85,B 0,C 180,E1 28148.772,E2 28148.772} C_VEL
LIN {X 0,Y 619.496,Z 1102.8,A -85,B 0,C 180,E1 28146.909,E2 28146.909} C_VEL
LIN {X 0,Y 620.79,Z 1088.273,A -85,B 0,C 180,E1 28144.837,E2 28144.837} C_VEL
LIN {X 0,Y 622.707,Z 1068.948,A -85,B 0,C 180,E1 28142.419,E2 28142.419} C_VEL
LIN {X 0,Y 624.537,Z 1051.517,A -85,B 0,C 180,E1 28140.497,E2 28140.497} C_VEL
LIN {X 0,Y 626.812,Z 1031.286,A -85,B 0,C 180,E1 28138.507,E2 28138.507} C_VEL
LIN {X 0,Y 629.352,Z 1008.218,A -85,B 0,C 180,E1 28136.523,E2 28136.523} C_VEL
LIN {X 0,Y 631.724,Z 987.178,A -85,B 0,C 180,E1 28134.934,E2 28134.934} C_VEL
LIN {X 0,Y 634.063,Z 966.163,A -85,B 0,C 180,E1 28133.524,E2 28133.524} C_VEL
LIN {X 0,Y 636.797,Z 940.246,A -85,B 0,C 180,E1 28132.013,E2 28132.013} C_VEL
LIN {X 0,Y 639.035,Z 917.01,A -85,B 0,C 180,E1 28130.852,E2 28130.852} C_VEL
LIN {X 0,Y 640.935,Z 896.096,A -85,B 0,C 180,E1 28129.947,E2 28129.947} C_VEL
LIN {X 0,Y 642.572,Z 875.969,A -85,B 0,C 180,E1 28129.192,E2 28129.192} C_VEL
LIN {X 0,Y 644.129,Z 854.754,A -85,B 0,C 180,E1 28128.515,E2 28128.515} C_VEL
LIN {X 0,Y 645.582,Z 831.763,A -85,B 0,C 180,E1 28127.912,E2 28127.912} C_VEL
LIN {X 0,Y 647.004,Z 803.34,A -85,B 0,C 180,E1 28127.344,E2 28127.344} C_VEL
LIN {X 0,Y 648.135,Z 757.965,A -85,B 0,C 180,E1 28126.713,E2 28126.713} C_VEL
LIN {X 0,Y 652.368,Z 541.338,A -85,B 0,C 180,E1 28123.811,E2 28123.811} C_VEL
LIN {X 0,Y 655.931,Z 380.352,A -85,B 0,C 180,E1 28121.567,E2 28121.567} C_VEL
LIN {X 0,Y 648.131,Z 369.227,A -85,B 0,C 180,E1 28120.591,E2 28120.591} C_VEL
LIN {X 0,Y 637.452,Z 358.863,A -85,B 0,C 180,E1 28119.266,E2 28119.266} C_VEL
LIN {X 0,Y 631.55,Z 353.114,A -85,B 0,C 180,E1 28118.478,E2 28118.478} C_VEL
LIN {X 0,Y 629.434,Z 349.167,A -85,B 0,C 180,E1 28117.475,E2 28117.475} C_VEL
LIN {X 0,Y 626.552,Z 344.141,A -85,B 0,C 180,E1 28116.077,E2 28116.077} C_VEL
LIN {X 0,Y 623.639,Z 339.217,A -85,B 0,C 180,E1 28114.581,E2 28114.581} C_VEL
LIN {X 0,Y 622.955,Z 337.859,A -85,B 0,C 180,E1 28114.179,E2 28114.179} C_VEL
LIN {X 0,Y 620.7,Z 334.473,A -85,B 0,C 180,E1 28112.99,E2 28112.99} C_VEL
LIN {X 0,Y 620.039,Z 332.688,A -85,B 0,C 180,E1 28112.48,E2 28112.48} C_VEL
LIN {X 0,Y 617.652,Z 329.642,A -85,B 0,C 180,E1 28111.201,E2 28111.201} C_VEL
LIN {X 0,Y 616.985,Z 327.351,A -85,B 0,C 180,E1 28110.481,E2 28110.481} C_VEL
LIN {X 0,Y 617.019,Z 327.372,A -85,B 0,C 180,E1 28107.297,E2 28107.297} C_VEL
LIN {X 0,Y 617.006,Z 327.339,A -85,B 0,C 180,E1 28104.002,E2 28104.002} C_VEL
LIN {X 0,Y 617.01,Z 327.335,A -85,B 0,C 180,E1 28100.769,E2 28100.769} C_VEL
LIN {X 0,Y 616.993,Z 327.379,A -85,B 0,C 180,E1 28097.641,E2 28097.641} C_VEL
LIN {X 0,Y 617.004,Z 327.345,A -85,B 0,C 180,E1 28094.452,E2 28094.452} C_VEL
LIN {X 0,Y 616.989,Z 327.335,A -85,B 0,C 180,E1 28091.356,E2 28091.356} C_VEL
LIN {X 0,Y 616.988,Z 327.377,A -85,B 0,C 180,E1 28088.199,E2 28088.199} C_VEL
LIN {X 0,Y 617.011,Z 327.342,A -85,B 0,C 180,E1 28085.114,E2 28085.114} C_VEL
LIN {X 0,Y 617.005,Z 327.331,A -85,B 0,C 180,E1 28081.764,E2 28081.764} C_VEL
LIN {X 0,Y 617.012,Z 327.348,A -85,B 0,C 180,E1 28078.514,E2 28078.514} C_VEL
LIN {X 0,Y 617.009,Z 327.527,A -85,B 0,C 180,E1 28077.678,E2 28077.678} C_VEL
LIN {X 0,Y 618.436,Z 330.993,A -85,B 0,C 180,E1 28076.57,E2 28076.57} C_VEL
LIN {X 0,Y 620.339,Z 333.028,A -85,B 0,C 180,E1 28075.655,E2 28075.655} C_VEL
LIN {X 0,Y 621.82,Z 336.531,A -85,B 0,C 180,E1 28074.649,E2 28074.649} C_VEL
LIN {X 0,Y 623.613,Z 338.695,A -85,B 0,C 180,E1 28073.833,E2 28073.833} C_VEL
LIN {X 0,Y 625.351,Z 342.34,A -85,B 0,C 180,E1 28072.836,E2 28072.836} C_VEL
LIN {X 0,Y 626.637,Z 343.913,A -85,B 0,C 180,E1 28072.297,E2 28072.297} C_VEL
LIN {X 0,Y 628.549,Z 347.744,A -85,B 0,C 180,E1 28071.308,E2 28071.308} C_VEL
LIN {X 0,Y 629.802,Z 349.624,A -85,B 0,C 180,E1 28070.773,E2 28070.773} C_VEL
LIN {X 0,Y 632.235,Z 353.763,A -85,B 0,C 180,E1 28069.705,E2 28069.705} C_VEL
LIN {X 0,Y 635.84,Z 360.708,A -85,B 0,C 180,E1 28068.112,E2 28068.112} C_VEL
LIN {X 0,Y 638.673,Z 365.843,A -85,B 0,C 180,E1 28066.971,E2 28066.971} C_VEL
LIN {X 0,Y 643.199,Z 374.275,A -85,B 0,C 180,E1 28065.229,E2 28065.229} C_VEL
LIN {X 0,Y 649.671,Z 386.762,A -85,B 0,C 180,E1 28062.887,E2 28062.887} C_VEL
LIN {X 0,Y 655.442,Z 398.53,A -85,B 0,C 180,E1 28060.9,E2 28060.9} C_VEL
LIN {X 0,Y 652.441,Z 429.313,A -85,B 0,C 180,E1 28058.372,E2 28058.372} C_VEL
LIN {X 0,Y 649.226,Z 464.388,A -85,B 0,C 180,E1 28055.622,E2 28055.622} C_VEL
LIN {X 0,Y 645.667,Z 505.837,A -85,B 0,C 180,E1 28052.517,E2 28052.517} C_VEL
LIN {X 0,Y 642.441,Z 546.209,A -85,B 0,C 180,E1 28049.614,E2 28049.614} C_VEL
LIN {X 0,Y 641.274,Z 568.816,A -85,B 0,C 180,E1 28047.985,E2 28047.985} C_VEL
LIN {X 0,Y 642.221,Z 584.04,A -85,B 0,C 180,E1 28046.767,E2 28046.767} C_VEL
LIN {X 0,Y 644.961,Z 597.527,A -85,B 0,C 180,E1 28045.561,E2 28045.561} C_VEL
LIN {X 0,Y 649.325,Z 609.215,A -85,B 0,C 180,E1 28044.393,E2 28044.393} C_VEL
LIN {X 0,Y 655.673,Z 620.036,A -85,B 0,C 180,E1 28043.179,E2 28043.179} C_VEL
LIN {X 0,Y 663.35,Z 628.909,A -85,B 0,C 180,E1 28042.048,E2 28042.048} C_VEL
LIN {X 0,Y 672.097,Z 636.111,A -85,B 0,C 180,E1 28041.001,E2 28041.001} C_VEL
LIN {X 0,Y 682.463,Z 642.142,A -85,B 0,C 180,E1 28039.97,E2 28039.97} C_VEL
LIN {X 0,Y 693.658,Z 646.489,A -85,B 0,C 180,E1 28039.014,E2 28039.014} C_VEL
LIN {X 0,Y 697.699,Z 646.925,A -85,B 0,C 180,E1 28038.539,E2 28038.539} C_VEL
LIN {X 0,Y 700.224,Z 646.231,A -85,B 0,C 180,E1 28038.065,E2 28038.065} C_VEL
LIN {X 0,Y 701.515,Z 644.581,A -85,B 0,C 180,E1 28037.586,E2 28037.586} C_VEL
LIN {X 0,Y 701.523,Z 641.954,A -85,B 0,C 180,E1 28037.103,E2 28037.103} C_VEL
LIN {X 0,Y 700.007,Z 638.382,A -85,B 0,C 180,E1 28036.638,E2 28036.638} C_VEL
LIN {X 0,Y 697.041,Z 634.21,A -85,B 0,C 180,E1 28036.256,E2 28036.256} C_VEL
LIN {X 0,Y 689.197,Z 624.615,A -85,B 0,C 180,E1 28035.624,E2 28035.624} C_VEL
LIN {X 0,Y 686.032,Z 638.262,A -85,B 0,C 180,E1 28035.365,E2 28035.365} C_VEL
LIN {X 0,Y 684.411,Z 643.609,A -85,B 0,C 180,E1 28035.231,E2 28035.231} C_VEL
LIN {X 0,Y 680.94,Z 674.303,A -85,B 0,C 180,E1 28034.977,E2 28034.977} C_VEL
LIN {X 0,Y 676.971,Z 692.392,A -85,B 0,C 180,E1 28034.879,E2 28034.879} C_VEL
LIN {X 0,Y 671.468,Z 709.271,A -85,B 0,C 180,E1 28034.775,E2 28034.775} C_VEL
LIN {X 0,Y 667.203,Z 719.785,A -85,B 0,C 180,E1 28034.594,E2 28034.594} C_VEL
LIN {X 0,Y 665.17,Z 724.518,A -85,B 0,C 180,E1 28034.464,E2 28034.464} C_VEL
LIN {X 0,Y 659.938,Z 736.386,A -85,B 0,C 180,E1 28034.363,E2 28034.363} C_VEL
LIN {X 0,Y 655.533,Z 745.988,A -85,B 0,C 180,E1 28034.129,E2 28034.129} C_VEL
LIN {X 0,Y 653.351,Z 750.917,A -85,B 0,C 180,E1 28033.948,E2 28033.948} C_VEL
LIN {X 0,Y 649.69,Z 758.934,A -85,B 0,C 180,E1 28033.709,E2 28033.709} C_VEL
LIN {X 0,Y 648.632,Z 761.984,A -85,B 0,C 180,E1 28033.588,E2 28033.588} C_VEL
LIN {X 0,Y 647.108,Z 830.303,A -85,B 0,C 180,E1 28032.659,E2 28032.659} C_VEL
LIN {X 0,Y 645.827,Z 857.678,A -85,B 0,C 180,E1 28032.137,E2 28032.137} C_VEL
LIN {X 0,Y 644.23,Z 883.888,A -85,B 0,C 180,E1 28031.469,E2 28031.469} C_VEL
LIN {X 0,Y 642.349,Z 909.427,A -85,B 0,C 180,E1 28030.648,E2 28030.648} C_VEL
LIN {X 0,Y 640.214,Z 934.856,A -85,B 0,C 180,E1 28029.648,E2 28029.648} C_VEL
LIN {X 0,Y 637.826,Z 959.788,A -85,B 0,C 180,E1 28028.486,E2 28028.486} C_VEL
LIN {X 0,Y 635.353,Z 983.916,A -85,B 0,C 180,E1 28027.178,E2 28027.178} C_VEL
LIN {X 0,Y 632.775,Z 1007.941,A -85,B 0,C 180,E1 28025.666,E2 28025.666} C_VEL
LIN {X 0,Y 630.371,Z 1029.636,A -85,B 0,C 180,E1 28024.106,E2 28024.106} C_VEL
LIN {X 0,Y 627.907,Z 1051.22,A -85,B 0,C 180,E1 28022.346,E2 28022.346} C_VEL
LIN {X 0,Y 625.471,Z 1073.119,A -85,B 0,C 180,E1 28020.316,E2 28020.316} C_VEL
LIN {X 0,Y 623.421,Z 1092.362,A -85,B 0,C 180,E1 28018.293,E2 28018.293} C_VEL
LIN {X 0,Y 621.63,Z 1109.513,A -85,B 0,C 180,E1 28016.251,E2 28016.251} C_VEL
LIN {X 0,Y 620.244,Z 1124.423,A -85,B 0,C 180,E1 28014.271,E2 28014.271} C_VEL
LIN {X 0,Y 618.902,Z 1140.157,A -85,B 0,C 180,E1 28011.912,E2 28011.912} C_VEL
LIN {X 0,Y 617.889,Z 1153.747,A -85,B 0,C 180,E1 28009.569,E2 28009.569} C_VEL
LIN {X 0,Y 617.181,Z 1164.753,A -85,B 0,C 180,E1 28007.4,E2 28007.4} C_VEL
LIN {X 0,Y 616.632,Z 1175.531,A -85,B 0,C 180,E1 28004.94,E2 28004.94} C_VEL
LIN {X 0,Y 616.245,Z 1184.901,A -85,B 0,C 180,E1 28002.366,E2 28002.366} C_VEL
LIN {X 0,Y 616.056,Z 1192.148,A -85,B 0,C 180,E1 27999.905,E2 27999.905} C_VEL
LIN {X 0,Y 615.96,Z 1197.724,A -85,B 0,C 180,E1 27997.46,E2 27997.46} C_VEL
LIN {X 0,Y 615.925,Z 1201.664,A -85,B 0,C 180,E1 27995.028,E2 27995.028} C_VEL
LIN {X 0,Y 615.909,Z 1204.093,A -85,B 0,C 180,E1 27992.604,E2 27992.604} C_VEL
LIN {X 0,Y 615.907,Z 1204.986,A -85,B 0,C 180,E1 27990.092,E2 27990.092} C_VEL
LIN {X 0,Y 615.909,Z 1204.204,A -85,B 0,C 180,E1 27987.58,E2 27987.58} C_VEL
LIN {X 0,Y 615.919,Z 1201.908,A -85,B 0,C 180,E1 27985.156,E2 27985.156} C_VEL
LIN {X 0,Y 615.962,Z 1197.996,A -85,B 0,C 180,E1 27982.676,E2 27982.676} C_VEL
LIN {X 0,Y 616.045,Z 1192.629,A -85,B 0,C 180,E1 27980.281,E2 27980.281} C_VEL
LIN {X 0,Y 616.221,Z 1185.509,A -85,B 0,C 180,E1 27977.822,E2 27977.822} C_VEL
LIN {X 0,Y 616.585,Z 1176.682,A -85,B 0,C 180,E1 27975.345,E2 27975.345} C_VEL
LIN {X 0,Y 617.138,Z 1165.486,A -85,B 0,C 180,E1 27972.752,E2 27972.752} C_VEL
LIN {X 0,Y 617.85,Z 1154.256,A -85,B 0,C 180,E1 27970.525,E2 27970.525} C_VEL
LIN {X 0,Y 618.853,Z 1140.748,A -85,B 0,C 180,E1 27968.184,E2 27968.184} C_VEL
LIN {X 0,Y 620.182,Z 1125.117,A -85,B 0,C 180,E1 27965.825,E2 27965.825} C_VEL
LIN {X 0,Y 621.562,Z 1110.274,A -85,B 0,C 180,E1 27963.846,E2 27963.846} C_VEL
LIN {X 0,Y 623.42,Z 1092.363,A -85,B 0,C 180,E1 27961.707,E2 27961.707} C_VEL
LIN {X 0,Y 625.471,Z 1073.119,A -85,B 0,C 180,E1 27959.685,E2 27959.685} C_VEL
LIN {X 0,Y 627.844,Z 1051.775,A -85,B 0,C 180,E1 27957.702,E2 27957.702} C_VEL
LIN {X 0,Y 630.297,Z 1030.299,A -85,B 0,C 180,E1 27955.944,E2 27955.944} C_VEL
LIN {X 0,Y 632.698,Z 1008.636,A -85,B 0,C 180,E1 27954.382,E2 27954.382} C_VEL
LIN {X 0,Y 635.265,Z 984.724,A -85,B 0,C 180,E1 27952.87,E2 27952.87} C_VEL
LIN {X 0,Y 637.729,Z 960.736,A -85,B 0,C 180,E1 27951.561,E2 27951.561} C_VEL
LIN {X 0,Y 640.099,Z 936.16,A -85,B 0,C 180,E1 27950.406,E2 27950.406} C_VEL
LIN {X 0,Y 642.303,Z 910.09,A -85,B 0,C 180,E1 27949.375,E2 27949.375} C_VEL
LIN {X 0,Y 644.219,Z 884.015,A -85,B 0,C 180,E1 27948.534,E2 27948.534} C_VEL
LIN {X 0,Y 645.816,Z 857.869,A -85,B 0,C 180,E1 27947.867,E2 27947.867} C_VEL
LIN {X 0,Y 647.097,Z 830.602,A -85,B 0,C 180,E1 27947.346,E2 27947.346} C_VEL
LIN {X 0,Y 648.548,Z 766.246,A -85,B 0,C 180,E1 27946.468,E2 27946.468} C_VEL
LIN {X 0,Y 649.454,Z 729.531,A -85,B 0,C 180,E1 27945.962,E2 27945.962} C_VEL
LIN {X 0,Y 656.334,Z 658.338,A -85,B 0,C 180,E1 27944.701,E2 27944.701} C_VEL
LIN {X 0,Y 657.782,Z 643.201,A -85,B 0,C 180,E1 27944.452,E2 27944.452} C_VEL
LIN {X 0,Y 660.551,Z 611.852,A -85,B 0,C 180,E1 27943.932,E2 27943.932} C_VEL
LIN {X 0,Y 662.611,Z 592.152,A -85,B 0,C 180,E1 27943.649,E2 27943.649} C_VEL
LIN {X 0,Y 664.406,Z 567.319,A -85,B 0,C 180,E1 27943.231,E2 27943.231} C_VEL
LIN {X 0,Y 668.125,Z 533.958,A -85,B 0,C 180,E1 27942.785,E2 27942.785} C_VEL
LIN {X 0,Y 669.385,Z 513.568,A -85,B 0,C 180,E1 27942.426,E2 27942.426} C_VEL
LIN {X 0,Y 673.03,Z 482.071,A -85,B 0,C 180,E1 27942.019,E2 27942.019} C_VEL
LIN {X 0,Y 674.436,Z 470.9,A -85,B 0,C 180,E1 27941.885,E2 27941.885} C_VEL
LIN {X 0,Y 675.22,Z 454.243,A -85,B 0,C 180,E1 27941.569,E2 27941.569} C_VEL
LIN {X 0,Y 678.349,Z 426.231,A -85,B 0,C 180,E1 27941.198,E2 27941.198} C_VEL
LIN {X 0,Y 681.54,Z 404.525,A -85,B 0,C 180,E1 27940.98,E2 27940.98} C_VEL
LIN {X 0,Y 672.775,Z 399.547,A -85,B 0,C 180,E1 27940.056,E2 27940.056} C_VEL
LIN {X 0,Y 665.247,Z 392.976,A -85,B 0,C 180,E1 27939.172,E2 27939.172} C_VEL
LIN {X 0,Y 657.924,Z 385.021,A -85,B 0,C 180,E1 27938.238,E2 27938.238} C_VEL
LIN {X 0,Y 643.478,Z 364.213,A -85,B 0,C 180,E1 27936.136,E2 27936.136} C_VEL
LIN {X 0,Y 635.91,Z 353.819,A -85,B 0,C 180,E1 27934.969,E2 27934.969} C_VEL
LIN {X 0,Y 632.327,Z 348.93,A -85,B 0,C 180,E1 27934.397,E2 27934.397} C_VEL
LIN {X 0,Y 628.797,Z 344.113,A -85,B 0,C 180,E1 27933.818,E2 27933.818} C_VEL
LIN {X 0,Y 625.711,Z 339.825,A -85,B 0,C 180,E1 27933.298,E2 27933.298} C_VEL
LIN {X 0,Y 622.012,Z 335.327,A -85,B 0,C 180,E1 27932.679,E2 27932.679} C_VEL
LIN {X 0,Y 620.984,Z 333.29,A -85,B 0,C 180,E1 27932.479,E2 27932.479} C_VEL
LIN {X 0,Y 618.28,Z 330.789,A -85,B 0,C 180,E1 27932.036,E2 27932.036} C_VEL
LIN {X 0,Y 617.031,Z 327.675,A -85,B 0,C 180,E1 27931.766,E2 27931.766} C_VEL
LIN {X 0,Y 616.979,Z 327.314,A -85,B 0,C 180,E1 27931.698,E2 27931.698} C_VEL
LIN {X 0,Y 617.013,Z 327.379,A -85,B 0,C 180,E1 27928.665,E2 27928.665} C_VEL
LIN {X 0,Y 616.972,Z 327.31,A -85,B 0,C 180,E1 27925.485,E2 27925.485} C_VEL
LIN {X 0,Y 616.99,Z 327.379,A -85,B 0,C 180,E1 27922.486,E2 27922.486} C_VEL
LIN {X 0,Y 616.996,Z 327.374,A -85,B 0,C 180,E1 27919.404,E2 27919.404} C_VEL
LIN {X 0,Y 616.997,Z 327.368,A -85,B 0,C 180,E1 27916.282,E2 27916.282} C_VEL
LIN {X 0,Y 617.019,Z 327.436,A -85,B 0,C 180,E1 27913.459,E2 27913.459} C_VEL
LIN {X 0,Y 620.785,Z 340.61,A -85,B 0,C 180,E1 27912.895,E2 27912.895} C_VEL
LIN {X 0,Y 620.79,Z 417.754,A -85,B 0,C 180,E1 27910.223,E2 27910.223} C_VEL
LIN {X 0,Y 621.174,Z 498.177,A -85,B 0,C 180,E1 27907.306,E2 27907.306} C_VEL
LIN {X 0,Y 621.261,Z 568.672,A -85,B 0,C 180,E1 27904.662,E2 27904.662} C_VEL
LIN {X 0,Y 620.972,Z 633.278,A -85,B 0,C 180,E1 27902.169,E2 27902.169} C_VEL
LIN {X 0,Y 620.351,Z 714.985,A -85,B 0,C 180,E1 27898.984,E2 27898.984} C_VEL
LIN {X 0,Y 619.551,Z 793.876,A -85,B 0,C 180,E1 27895.835,E2 27895.835} C_VEL
LIN {X 0,Y 618.831,Z 846.134,A -85,B 0,C 180,E1 27893.739,E2 27893.739} C_VEL
LIN {X 0,Y 618.601,Z 850.358,A -85,B 0,C 180,E1 27893.605,E2 27893.605} C_VEL
LIN {X 0,Y 618.101,Z 964.383,A -85,B 0,C 180,E1 27892.225,E2 27892.225} C_VEL
LIN {X 0,Y 618.093,Z 976.731,A -85,B 0,C 180,E1 27891.953,E2 27891.953} C_VEL
LIN {X 0,Y 618.047,Z 988.358,A -85,B 0,C 180,E1 27891.581,E2 27891.581} C_VEL
LIN {X 0,Y 617.943,Z 1001.108,A -85,B 0,C 180,E1 27891.032,E2 27891.032} C_VEL
LIN {X 0,Y 617.736,Z 1014.261,A -85,B 0,C 180,E1 27890.262,E2 27890.262} C_VEL
LIN {X 0,Y 617.572,Z 1023.813,A -85,B 0,C 180,E1 27889.552,E2 27889.552} C_VEL
LIN {X 0,Y 617.388,Z 1032.219,A -85,B 0,C 180,E1 27888.793,E2 27888.793} C_VEL
LIN {X 0,Y 617.209,Z 1040.021,A -85,B 0,C 180,E1 27887.937,E2 27887.937} C_VEL
LIN {X 0,Y 617.032,Z 1047.775,A -85,B 0,C 180,E1 27886.884,E2 27886.884} C_VEL
LIN {X 0,Y 616.853,Z 1054.685,A -85,B 0,C 180,E1 27885.64,E2 27885.64} C_VEL
LIN {X 0,Y 616.755,Z 1059.036,A -85,B 0,C 180,E1 27884.581,E2 27884.581} C_VEL
LIN {X 0,Y 616.682,Z 1062.175,A -85,B 0,C 180,E1 27883.516,E2 27883.516} C_VEL
LIN {X 0,Y 616.642,Z 1064.17,A -85,B 0,C 180,E1 27882.446,E2 27882.446} C_VEL
LIN {X 0,Y 616.611,Z 1065.065,A -85,B 0,C 180,E1 27881.37,E2 27881.37} C_VEL
LIN {X 0,Y 616.609,Z 1064.773,A -85,B 0,C 180,E1 27880.141,E2 27880.141} C_VEL
LIN {X 0,Y 616.629,Z 1062.57,A -85,B 0,C 180,E1 27878.701,E2 27878.701} C_VEL
LIN {X 0,Y 616.679,Z 1059.127,A -85,B 0,C 180,E1 27877.502,E2 27877.502} C_VEL
LIN {X 0,Y 616.753,Z 1054.602,A -85,B 0,C 180,E1 27876.394,E2 27876.394} C_VEL
LIN {X 0,Y 616.907,Z 1047.997,A -85,B 0,C 180,E1 27875.179,E2 27875.179} C_VEL
LIN {X 0,Y 617.087,Z 1039.85,A -85,B 0,C 180,E1 27874.056,E2 27874.056} C_VEL
LIN {X 0,Y 617.272,Z 1031.43,A -85,B 0,C 180,E1 27873.132,E2 27873.132} C_VEL
LIN {X 0,Y 617.464,Z 1022.733,A -85,B 0,C 180,E1 27872.349,E2 27872.349} C_VEL
LIN {X 0,Y 617.651,Z 1012.277,A -85,B 0,C 180,E1 27871.579,E2 27871.579} C_VEL
LIN {X 0,Y 617.88,Z 998.644,A -85,B 0,C 180,E1 27870.799,E2 27870.799} C_VEL
LIN {X 0,Y 618.015,Z 986.388,A -85,B 0,C 180,E1 27870.277,E2 27870.277} C_VEL
LIN {X 0,Y 618.093,Z 974.577,A -85,B 0,C 180,E1 27869.901,E2 27869.901} C_VEL
LIN {X 0,Y 618.105,Z 972.983,A -85,B 0,C 180,E1 27869.858,E2 27869.858} C_VEL
LIN {X 0,Y 617.414,Z 966.606,A -85,B 0,C 180,E1 27869.693,E2 27869.693} C_VEL
LIN {X 0,Y 613.148,Z 953.07,A -85,B 0,C 180,E1 27869.403,E2 27869.403} C_VEL
LIN {X 0,Y 610.655,Z 943.492,A -85,B 0,C 180,E1 27869.247,E2 27869.247} C_VEL
LIN {X 0,Y 610.318,Z 939.106,A -85,B 0,C 180,E1 27869.191,E2 27869.191} C_VEL
LIN {X 0,Y 610.908,Z 846.666,A -85,B 0,C 180,E1 27868.057,E2 27868.057} C_VEL
LIN {X 0,Y 611.87,Z 788.245,A -85,B 0,C 180,E1 27865.647,E2 27865.647} C_VEL
LIN {X 0,Y 613.038,Z 706.966,A -85,B 0,C 180,E1 27862.285,E2 27862.285} C_VEL
LIN {X 0,Y 614.175,Z 628.934,A -85,B 0,C 180,E1 27859.061,E2 27859.061} C_VEL
LIN {X 0,Y 614.495,Z 610.492,A -85,B 0,C 180,E1 27858.278,E2 27858.278} C_VEL
LIN {X 0,Y 615.701,Z 612.392,A -85,B 0,C 180,E1 27858.129,E2 27858.129} C_VEL
LIN {X 0,Y 617.468,Z 612.502,A -85,B 0,C 180,E1 27857.964,E2 27857.964} C_VEL
LIN {X 0,Y 620.199,Z 610.405,A -85,B 0,C 180,E1 27857.756,E2 27857.756} C_VEL
LIN {X 0,Y 623.65,Z 605.315,A -85,B 0,C 180,E1 27857.539,E2 27857.539} C_VEL
LIN {X 0,Y 624.226,Z 604.469,A -85,B 0,C 180,E1 27857.502,E2 27857.502} C_VEL
LIN {X 0,Y 627.78,Z 603.21,A -85,B 0,C 180,E1 27857.211,E2 27857.211} C_VEL
LIN {X 0,Y 631.67,Z 599.816,A -85,B 0,C 180,E1 27856.934,E2 27856.934} C_VEL
LIN {X 0,Y 635.1,Z 595.278,A -85,B 0,C 180,E1 27856.713,E2 27856.713} C_VEL
LIN {X 0,Y 639.687,Z 592.512,A -85,B 0,C 180,E1 27856.367,E2 27856.367} C_VEL
LIN {X 0,Y 644.352,Z 587.53,A -85,B 0,C 180,E1 27856.057,E2 27856.057} C_VEL
LIN {X 0,Y 645.595,Z 586.024,A -85,B 0,C 180,E1 27855.978,E2 27855.978} C_VEL
LIN {X 0,Y 642.725,Z 737.741,A -85,B 0,C 180,E1 27853.959,E2 27853.959} C_VEL
LIN {X 0,Y 641.235,Z 799.276,A -85,B 0,C 180,E1 27853.114,E2 27853.114} C_VEL
LIN {X 0,Y 639.962,Z 826.671,A -85,B 0,C 180,E1 27852.603,E2 27852.603} C_VEL
LIN {X 0,Y 638.199,Z 853.163,A -85,B 0,C 180,E1 27851.923,E2 27851.923} C_VEL
LIN {X 0,Y 636.567,Z 874.431,A -85,B 0,C 180,E1 27851.249,E2 27851.249} C_VEL
LIN {X 0,Y 634.862,Z 894.124,A -85,B 0,C 180,E1 27850.518,E2 27850.518} C_VEL
LIN {X 0,Y 632.843,Z 915.261,A -85,B 0,C 180,E1 27849.608,E2 27849.608} C_VEL
LIN {X 0,Y 630.744,Z 935.701,A -85,B 0,C 180,E1 27848.599,E2 27848.599} C_VEL
LIN {X 0,Y 628.283,Z 958.277,A -85,B 0,C 180,E1 27847.327,E2 27847.327} C_VEL
LIN {X 0,Y 625.406,Z 983.338,A -85,B 0,C 180,E1 27845.69,E2 27845.69} C_VEL
LIN {X 0,Y 622.965,Z 1003.579,A -85,B 0,C 180,E1 27844.179,E2 27844.179} C_VEL
LIN {X 0,Y 620.551,Z 1023.567,A -85,B 0,C 180,E1 27842.505,E2 27842.505} C_VEL
LIN {X 0,Y 618.092,Z 1044.485,A -85,B 0,C 180,E1 27840.529,E2 27840.529} C_VEL
LIN {X 0,Y 615.808,Z 1064.136,A -85,B 0,C 180,E1 27838.409,E2 27838.409} C_VEL
LIN {X 0,Y 614.055,Z 1079.937,A -85,B 0,C 180,E1 27836.499,E2 27836.499} C_VEL
LIN {X 0,Y 612.649,Z 1094.078,A -85,B 0,C 180,E1 27834.594,E2 27834.594} C_VEL
LIN {X 0,Y 611.182,Z 1110.016,A -85,B 0,C 180,E1 27832.184,E2 27832.184} C_VEL
LIN {X 0,Y 610.118,Z 1122.921,A -85,B 0,C 180,E1 27829.931,E2 27829.931} C_VEL
LIN {X 0,Y 609.401,Z 1132.913,A -85,B 0,C 180,E1 27827.968,E2 27827.968} C_VEL
LIN {X 0,Y 608.885,Z 1141.695,A -85,B 0,C 180,E1 27826.016,E2 27826.016} C_VEL
LIN {X 0,Y 608.497,Z 1149.341,A -85,B 0,C 180,E1 27824.076,E2 27824.076} C_VEL
LIN {X 0,Y 608.218,Z 1156.539,A -85,B 0,C 180,E1 27821.956,E2 27821.956} C_VEL
LIN {X 0,Y 608.047,Z 1163.205,A -85,B 0,C 180,E1 27819.561,E2 27819.561} C_VEL
LIN {X 0,Y 607.947,Z 1168.867,A -85,B 0,C 180,E1 27816.897,E2 27816.897} C_VEL
LIN {X 0,Y 607.915,Z 1172.404,A -85,B 0,C 180,E1 27814.435,E2 27814.435} C_VEL
LIN {X 0,Y 607.909,Z 1174.318,A -85,B 0,C 180,E1 27812.169,E2 27812.169} C_VEL
LIN {X 0,Y 607.897,Z 1174.938,A -85,B 0,C 180,E1 27809.718,E2 27809.718} C_VEL
LIN {X 0,Y 607.907,Z 1174.111,A -85,B 0,C 180,E1 27807.362,E2 27807.362} C_VEL
LIN {X 0,Y 607.924,Z 1171.503,A -85,B 0,C 180,E1 27804.716,E2 27804.716} C_VEL
LIN {X 0,Y 607.964,Z 1167.399,A -85,B 0,C 180,E1 27802.251,E2 27802.251} C_VEL
LIN {X 0,Y 608.066,Z 1162.212,A -85,B 0,C 180,E1 27799.963,E2 27799.963} C_VEL
LIN {X 0,Y 608.24,Z 1155.926,A -85,B 0,C 180,E1 27797.758,E2 27797.758} C_VEL
LIN {X 0,Y 608.528,Z 1148.613,A -85,B 0,C 180,E1 27795.636,E2 27795.636} C_VEL
LIN {X 0,Y 608.974,Z 1140.032,A -85,B 0,C 180,E1 27793.499,E2 27793.499} C_VEL
LIN {X 0,Y 609.794,Z 1127.374,A -85,B 0,C 180,E1 27790.818,E2 27790.818} C_VEL
LIN {X 0,Y 610.675,Z 1115.677,A -85,B 0,C 180,E1 27788.687,E2 27788.687} C_VEL
LIN {X 0,Y 611.687,Z 1104.092,A -85,B 0,C 180,E1 27786.801,E2 27786.801} C_VEL
LIN {X 0,Y 612.923,Z 1090.949,A -85,B 0,C 180,E1 27784.878,E2 27784.878} C_VEL
LIN {X 0,Y 614.617,Z 1075.094,A -85,B 0,C 180,E1 27782.799,E2 27782.799} C_VEL
LIN {X 0,Y 616.835,Z 1054.974,A -85,B 0,C 180,E1 27780.478,E2 27780.478} C_VEL
LIN {X 0,Y 619.008,Z 1036.545,A -85,B 0,C 180,E1 27778.607,E2 27778.607} C_VEL
LIN {X 0,Y 621.434,Z 1016.547,A -85,B 0,C 180,E1 27776.792,E2 27776.792} C_VEL
LIN {X 0,Y 624.243,Z 992.795,A -85,B 0,C 180,E1 27774.9,E2 27774.9} C_VEL
LIN {X 0,Y 626.739,Z 971.602,A -85,B 0,C 180,E1 27773.427,E2 27773.427} C_VEL
LIN {X 0,Y 629.038,Z 951.499,A -85,B 0,C 180,E1 27772.187,E2 27772.187} C_VEL
LIN {X 0,Y 631.327,Z 930.526,A -85,B 0,C 180,E1 27771.043,E2 27771.043} C_VEL
LIN {X 0,Y 633.959,Z 904.796,A -85,B 0,C 180,E1 27769.83,E2 27769.83} C_VEL
LIN {X 0,Y 636.128,Z 879.651,A -85,B 0,C 180,E1 27768.844,E2 27768.844} C_VEL
LIN {X 0,Y 637.835,Z 858.015,A -85,B 0,C 180,E1 27768.131,E2 27768.131} C_VEL
LIN {X 0,Y 639.267,Z 837.134,A -85,B 0,C 180,E1 27767.56,E2 27767.56} C_VEL
LIN {X 0,Y 640.463,Z 816.05,A -85,B 0,C 180,E1 27767.093,E2 27767.093} C_VEL
LIN {X 0,Y 641.399,Z 794.677,A -85,B 0,C 180,E1 27766.727,E2 27766.727} C_VEL
LIN {X 0,Y 644.612,Z 641.014,A -85,B 0,C 180,E1 27764.659,E2 27764.659} C_VEL
LIN {X 0,Y 647.403,Z 506.506,A -85,B 0,C 180,E1 27762.832,E2 27762.832} C_VEL
LIN {X 0,Y 650.54,Z 384.283,A -85,B 0,C 180,E1 27761.092,E2 27761.092} C_VEL
LIN {X 0,Y 643.87,Z 374.974,A -85,B 0,C 180,E1 27760.243,E2 27760.243} C_VEL
LIN {X 0,Y 633.695,Z 365.269,A -85,B 0,C 180,E1 27758.961,E2 27758.961} C_VEL
LIN {X 0,Y 628.163,Z 359.963,A -85,B 0,C 180,E1 27758.229,E2 27758.229} C_VEL
LIN {X 0,Y 625.511,Z 357.548,A -85,B 0,C 180,E1 27757.849,E2 27757.849} C_VEL
LIN {X 0,Y 623.953,Z 354.4,A -85,B 0,C 180,E1 27757.053,E2 27757.053} C_VEL
LIN {X 0,Y 621.766,Z 350.392,A -85,B 0,C 180,E1 27755.943,E2 27755.943} C_VEL
LIN {X 0,Y 619.019,Z 345.865,A -85,B 0,C 180,E1 27754.537,E2 27754.537} C_VEL
LIN {X 0,Y 618.376,Z 344.394,A -85,B 0,C 180,E1 27754.121,E2 27754.121} C_VEL
LIN {X 0,Y 615.999,Z 340.717,A -85,B 0,C 180,E1 27752.83,E2 27752.83} C_VEL
LIN {X 0,Y 615.278,Z 339.073,A -85,B 0,C 180,E1 27752.321,E2 27752.321} C_VEL
LIN {X 0,Y 613.005,Z 335.91,A -85,B 0,C 180,E1 27751.027,E2 27751.027} C_VEL
LIN {X 0,Y 612.167,Z 333.732,A -85,B 0,C 180,E1 27750.312,E2 27750.312} C_VEL
LIN {X 0,Y 609.569,Z 330.268,A -85,B 0,C 180,E1 27748.653,E2 27748.653} C_VEL
LIN {X 0,Y 609.047,Z 328.337,A -85,B 0,C 180,E1 27747.967,E2 27747.967} C_VEL
LIN {X 0,Y 609.053,Z 328.32,A -85,B 0,C 180,E1 27744.852,E2 27744.852} C_VEL
LIN {X 0,Y 609.068,Z 328.344,A -85,B 0,C 180,E1 27741.697,E2 27741.697} C_VEL
LIN {X 0,Y 609.064,Z 328.357,A -85,B 0,C 180,E1 27738.373,E2 27738.373} C_VEL
LIN {X 0,Y 609.066,Z 328.319,A -85,B 0,C 180,E1 27735.131,E2 27735.131} C_VEL
LIN {X 0,Y 609.059,Z 328.334,A -85,B 0,C 180,E1 27732.034,E2 27732.034} C_VEL
LIN {X 0,Y 609.072,Z 328.362,A -85,B 0,C 180,E1 27728.782,E2 27728.782} C_VEL
LIN {X 0,Y 609.047,Z 328.323,A -85,B 0,C 180,E1 27725.559,E2 27725.559} C_VEL
LIN {X 0,Y 609.068,Z 328.325,A -85,B 0,C 180,E1 27722.446,E2 27722.446} C_VEL
LIN {X 0,Y 609.08,Z 328.544,A -85,B 0,C 180,E1 27720.188,E2 27720.188} C_VEL
LIN {X 0,Y 610.508,Z 332.035,A -85,B 0,C 180,E1 27718.874,E2 27718.874} C_VEL
LIN {X 0,Y 612.505,Z 334.206,A -85,B 0,C 180,E1 27717.755,E2 27717.755} C_VEL
LIN {X 0,Y 614.136,Z 337.816,A -85,B 0,C 180,E1 27716.546,E2 27716.546} C_VEL
LIN {X 0,Y 615.786,Z 339.743,A -85,B 0,C 180,E1 27715.716,E2 27715.716} C_VEL
LIN {X 0,Y 617.516,Z 343.378,A -85,B 0,C 180,E1 27714.611,E2 27714.611} C_VEL
LIN {X 0,Y 619.038,Z 345.418,A -85,B 0,C 180,E1 27713.88,E2 27713.88} C_VEL
LIN {X 0,Y 621.057,Z 349.198,A -85,B 0,C 180,E1 27712.786,E2 27712.786} C_VEL
LIN {X 0,Y 622.037,Z 350.658,A -85,B 0,C 180,E1 27712.333,E2 27712.333} C_VEL
LIN {X 0,Y 624.254,Z 354.632,A -85,B 0,C 180,E1 27711.248,E2 27711.248} C_VEL
LIN {X 0,Y 627.98,Z 361.31,A -85,B 0,C 180,E1 27709.542,E2 27709.542} C_VEL
LIN {X 0,Y 630.834,Z 366.628,A -85,B 0,C 180,E1 27708.294,E2 27708.294} C_VEL
LIN {X 0,Y 635.441,Z 374.98,A -85,B 0,C 180,E1 27706.44,E2 27706.44} C_VEL
LIN {X 0,Y 642.553,Z 388.769,A -85,B 0,C 180,E1 27703.734,E2 27703.734} C_VEL
LIN {X 0,Y 649.708,Z 403.432,A -85,B 0,C 180,E1 27701.191,E2 27701.191} C_VEL
LIN {X 0,Y 646.882,Z 431.138,A -85,B 0,C 180,E1 27698.89,E2 27698.89} C_VEL
LIN {X 0,Y 643.448,Z 466.109,A -85,B 0,C 180,E1 27696.121,E2 27696.121} C_VEL
LIN {X 0,Y 639.728,Z 506.711,A -85,B 0,C 180,E1 27693.046,E2 27693.046} C_VEL
LIN {X 0,Y 636.231,Z 547.694,A -85,B 0,C 180,E1 27690.067,E2 27690.067} C_VEL
LIN {X 0,Y 634.836,Z 571.149,A -85,B 0,C 180,E1 27688.366,E2 27688.366} C_VEL
LIN {X 0,Y 635.608,Z 586.536,A -85,B 0,C 180,E1 27687.13,E2 27687.13} C_VEL
LIN {X 0,Y 638.197,Z 600.477,A -85,B 0,C 180,E1 27685.882,E2 27685.882} C_VEL
LIN {X 0,Y 642.747,Z 613.279,A -85,B 0,C 180,E1 27684.6,E2 27684.6} C_VEL
LIN {X 0,Y 648.839,Z 624.069,A -85,B 0,C 180,E1 27683.388,E2 27683.388} C_VEL
LIN {X 0,Y 656.338,Z 633.207,A -85,B 0,C 180,E1 27682.235,E2 27682.235} C_VEL
LIN {X 0,Y 665.502,Z 641.159,A -85,B 0,C 180,E1 27681.095,E2 27681.095} C_VEL
LIN {X 0,Y 676.389,Z 647.808,A -85,B 0,C 180,E1 27679.98,E2 27679.98} C_VEL
LIN {X 0,Y 689.057,Z 652.957,A -85,B 0,C 180,E1 27678.902,E2 27678.902} C_VEL
LIN {X 0,Y 693.449,Z 653.734,A -85,B 0,C 180,E1 27678.449,E2 27678.449} C_VEL
LIN {X 0,Y 696.31,Z 653.371,A -85,B 0,C 180,E1 27677.997,E2 27677.997} C_VEL
LIN {X 0,Y 698.167,Z 651.842,A -85,B 0,C 180,E1 27677.469,E2 27677.469} C_VEL
LIN {X 0,Y 698.491,Z 649.164,A -85,B 0,C 180,E1 27676.935,E2 27676.935} C_VEL
LIN {X 0,Y 697.225,Z 645.738,A -85,B 0,C 180,E1 27676.461,E2 27676.461} C_VEL
LIN {X 0,Y 694.531,Z 641.746,A -85,B 0,C 180,E1 27676.068,E2 27676.068} C_VEL
LIN {X 0,Y 691.972,Z 639.025,A -85,B 0,C 180,E1 27675.848,E2 27675.848} C_VEL
LIN {X 0,Y 689.923,Z 646.152,A -85,B 0,C 180,E1 27675.683,E2 27675.683} C_VEL
LIN {X 0,Y 687.572,Z 663.265,A -85,B 0,C 180,E1 27675.587,E2 27675.587} C_VEL
LIN {X 0,Y 683.279,Z 680.684,A -85,B 0,C 180,E1 27675.55,E2 27675.55} C_VEL
LIN {X 0,Y 676.872,Z 698.321,A -85,B 0,C 180,E1 27675.518,E2 27675.518} C_VEL
LIN {X 0,Y 670.243,Z 712.746,A -85,B 0,C 180,E1 27675.424,E2 27675.424} C_VEL
LIN {X 0,Y 665.478,Z 722.572,A -85,B 0,C 180,E1 27675.227,E2 27675.227} C_VEL
LIN {X 0,Y 663.851,Z 725.918,A -85,B 0,C 180,E1 27675.147,E2 27675.147} C_VEL
LIN {X 0,Y 657.321,Z 737.683,A -85,B 0,C 180,E1 27675.016,E2 27675.016} C_VEL
LIN {X 0,Y 652.411,Z 747.213,A -85,B 0,C 180,E1 27674.765,E2 27674.765} C_VEL
LIN {X 0,Y 649.697,Z 752.942,A -85,B 0,C 180,E1 27674.568,E2 27674.568} C_VEL
LIN {X 0,Y 645.724,Z 761.171,A -85,B 0,C 180,E1 27674.293,E2 27674.293} C_VEL
LIN {X 0,Y 642.696,Z 768.736,A -85,B 0,C 180,E1 27673.991,E2 27673.991} C_VEL
LIN {X 0,Y 641.21,Z 830.591,A -85,B 0,C 180,E1 27673.141,E2 27673.141} C_VEL
LIN {X 0,Y 639.858,Z 857.885,A -85,B 0,C 180,E1 27672.617,E2 27672.617} C_VEL
LIN {X 0,Y 638.185,Z 883.88,A -85,B 0,C 180,E1 27671.951,E2 27671.951} C_VEL
LIN {X 0,Y 636.2,Z 909.435,A -85,B 0,C 180,E1 27671.126,E2 27671.126} C_VEL
LIN {X 0,Y 634.032,Z 933.811,A -85,B 0,C 180,E1 27670.164,E2 27670.164} C_VEL
LIN {X 0,Y 631.634,Z 957.79,A -85,B 0,C 180,E1 27669.051,E2 27669.051} C_VEL
LIN {X 0,Y 629.197,Z 980.523,A -85,B 0,C 180,E1 27667.832,E2 27667.832} C_VEL
LIN {X 0,Y 626.306,Z 1005.634,A -85,B 0,C 180,E1 27666.271,E2 27666.271} C_VEL
LIN {X 0,Y 623.661,Z 1027.952,A -85,B 0,C 180,E1 27664.667,E2 27664.667} C_VEL
LIN {X 0,Y 621.139,Z 1048.88,A -85,B 0,C 180,E1 27662.961,E2 27662.961} C_VEL
LIN {X 0,Y 618.624,Z 1069.844,A -85,B 0,C 180,E1 27661.036,E2 27661.036} C_VEL
LIN {X 0,Y 616.47,Z 1088.267,A -85,B 0,C 180,E1 27659.115,E2 27659.115} C_VEL
LIN {X 0,Y 614.377,Z 1107.174,A -85,B 0,C 180,E1 27656.899,E2 27656.899} C_VEL
LIN {X 0,Y 612.799,Z 1122.41,A -85,B 0,C 180,E1 27654.876,E2 27654.876} C_VEL
LIN {X 0,Y 611.378,Z 1137.728,A -85,B 0,C 180,E1 27652.601,E2 27652.601} C_VEL
LIN {X 0,Y 610.168,Z 1152.23,A -85,B 0,C 180,E1 27650.118,E2 27650.118} C_VEL
LIN {X 0,Y 609.372,Z 1163.638,A -85,B 0,C 180,E1 27647.867,E2 27647.867} C_VEL
LIN {X 0,Y 608.727,Z 1174.586,A -85,B 0,C 180,E1 27645.376,E2 27645.376} C_VEL
LIN {X 0,Y 608.313,Z 1184.283,A -85,B 0,C 180,E1 27642.723,E2 27642.723} C_VEL
LIN {X 0,Y 608.084,Z 1191.661,A -85,B 0,C 180,E1 27640.228,E2 27640.228} C_VEL
LIN {X 0,Y 607.969,Z 1197.332,A -85,B 0,C 180,E1 27637.749,E2 27637.749} C_VEL
LIN {X 0,Y 607.927,Z 1201.415,A -85,B 0,C 180,E1 27635.284,E2 27635.284} C_VEL
LIN {X 0,Y 607.914,Z 1203.981,A -85,B 0,C 180,E1 27632.827,E2 27632.827} C_VEL
LIN {X 0,Y 607.892,Z 1204.916,A -85,B 0,C 180,E1 27630.47,E2 27630.47} C_VEL
LIN {X 0,Y 607.911,Z 1204.417,A -85,B 0,C 180,E1 27627.925,E2 27627.925} C_VEL
LIN {X 0,Y 607.915,Z 1202.393,A -85,B 0,C 180,E1 27625.471,E2 27625.471} C_VEL
LIN {X 0,Y 607.948,Z 1198.773,A -85,B 0,C 180,E1 27623.008,E2 27623.008} C_VEL
LIN {X 0,Y 608.04,Z 1193.558,A -85,B 0,C 180,E1 27620.534,E2 27620.534} C_VEL
LIN {X 0,Y 608.221,Z 1186.608,A -85,B 0,C 180,E1 27618.003,E2 27618.003} C_VEL
LIN {X 0,Y 608.55,Z 1178.477,A -85,B 0,C 180,E1 27615.634,E2 27615.634} C_VEL
LIN {X 0,Y 609.056,Z 1168.588,A -85,B 0,C 180,E1 27613.205,E2 27613.205} C_VEL
LIN {X 0,Y 609.867,Z 1156.329,A -85,B 0,C 180,E1 27610.658,E2 27610.658} C_VEL
LIN {X 0,Y 610.857,Z 1143.73,A -85,B 0,C 180,E1 27608.389,E2 27608.389} C_VEL
LIN {X 0,Y 612.144,Z 1129.244,A -85,B 0,C 180,E1 27606.102,E2 27606.102} C_VEL
LIN {X 0,Y 613.802,Z 1112.615,A -85,B 0,C 180,E1 27603.802,E2 27603.802} C_VEL
LIN {X 0,Y 615.453,Z 1097.145,A -85,B 0,C 180,E1 27601.891,E2 27601.891} C_VEL
LIN {X 0,Y 617.75,Z 1077.334,A -85,B 0,C 180,E1 27599.721,E2 27599.721} C_VEL
LIN {X 0,Y 620.035,Z 1058.028,A -85,B 0,C 180,E1 27597.847,E2 27597.847} C_VEL
LIN {X 0,Y 622.7,Z 1035.848,A -85,B 0,C 180,E1 27595.951,E2 27595.951} C_VEL
LIN {X 0,Y 625.432,Z 1013.006,A -85,B 0,C 180,E1 27594.244,E2 27594.244} C_VEL
LIN {X 0,Y 628.047,Z 990.657,A -85,B 0,C 180,E1 27592.772,E2 27592.772} C_VEL
LIN {X 0,Y 630.79,Z 965.725,A -85,B 0,C 180,E1 27591.35,E2 27591.35} C_VEL
LIN {X 0,Y 633.35,Z 940.74,A -85,B 0,C 180,E1 27590.136,E2 27590.136} C_VEL
LIN {X 0,Y 635.669,Z 915.463,A -85,B 0,C 180,E1 27589.099,E2 27589.099} C_VEL
LIN {X 0,Y 637.816,Z 888.6,A -85,B 0,C 180,E1 27588.19,E2 27588.19} C_VEL
LIN {X 0,Y 639.609,Z 862.182,A -85,B 0,C 180,E1 27587.481,E2 27587.481} C_VEL
LIN {X 0,Y 641.022,Z 835.844,A -85,B 0,C 180,E1 27586.943,E2 27586.943} C_VEL
LIN {X 0,Y 642.055,Z 800.32,A -85,B 0,C 180,E1 27586.433,E2 27586.433} C_VEL
LIN {X 0,Y 643.168,Z 755.326,A -85,B 0,C 180,E1 27585.812,E2 27585.812} C_VEL
LIN {X 0,Y 647.982,Z 696.285,A -85,B 0,C 180,E1 27584.799,E2 27584.799} C_VEL
LIN {X 0,Y 650.907,Z 659,A -85,B 0,C 180,E1 27584.188,E2 27584.188} C_VEL
LIN {X 0,Y 652.242,Z 643.567,A -85,B 0,C 180,E1 27583.946,E2 27583.946} C_VEL
LIN {X 0,Y 654.938,Z 611.322,A -85,B 0,C 180,E1 27583.432,E2 27583.432} C_VEL
LIN {X 0,Y 656.862,Z 592.605,A -85,B 0,C 180,E1 27583.165,E2 27583.165} C_VEL
LIN {X 0,Y 658.767,Z 566.999,A -85,B 0,C 180,E1 27582.736,E2 27582.736} C_VEL
LIN {X 0,Y 662.425,Z 534.48,A -85,B 0,C 180,E1 27582.3,E2 27582.3} C_VEL
LIN {X 0,Y 663.827,Z 513.187,A -85,B 0,C 180,E1 27581.927,E2 27581.927} C_VEL
LIN {X 0,Y 667.608,Z 481.201,A -85,B 0,C 180,E1 27581.516,E2 27581.516} C_VEL
LIN {X 0,Y 668.806,Z 471.533,A -85,B 0,C 180,E1 27581.397,E2 27581.397} C_VEL
LIN {X 0,Y 669.724,Z 454.064,A -85,B 0,C 180,E1 27581.069,E2 27581.069} C_VEL
LIN {X 0,Y 672.986,Z 425.527,A -85,B 0,C 180,E1 27580.694,E2 27580.694} C_VEL
LIN {X 0,Y 675.136,Z 410.192,A -85,B 0,C 180,E1 27580.529,E2 27580.529} C_VEL
LIN {X 0,Y 666.561,Z 404.398,A -85,B 0,C 180,E1 27579.58,E2 27579.58} C_VEL
LIN {X 0,Y 655.415,Z 393.214,A -85,B 0,C 180,E1 27578.188,E2 27578.188} C_VEL
LIN {X 0,Y 636.956,Z 366.686,A -85,B 0,C 180,E1 27575.454,E2 27575.454} C_VEL
LIN {X 0,Y 628.152,Z 354.799,A -85,B 0,C 180,E1 27574.05,E2 27574.05} C_VEL
LIN {X 0,Y 624.891,Z 350.372,A -85,B 0,C 180,E1 27573.507,E2 27573.507} C_VEL
LIN {X 0,Y 621.077,Z 345.263,A -85,B 0,C 180,E1 27572.857,E2 27572.857} C_VEL
LIN {X 0,Y 618.036,Z 341.121,A -85,B 0,C 180,E1 27572.324,E2 27572.324} C_VEL
LIN {X 0,Y 616.984,Z 339.762,A -85,B 0,C 180,E1 27572.139,E2 27572.139} C_VEL
LIN {X 0,Y 614.176,Z 336.352,A -85,B 0,C 180,E1 27571.643,E2 27571.643} C_VEL
LIN {X 0,Y 612.993,Z 334.24,A -85,B 0,C 180,E1 27571.41,E2 27571.41} C_VEL
LIN {X 0,Y 610.261,Z 331.624,A -85,B 0,C 180,E1 27570.935,E2 27570.935} C_VEL
LIN {X 0,Y 609.089,Z 328.509,A -85,B 0,C 180,E1 27570.663,E2 27570.663} C_VEL
LIN {X 0,Y 609.069,Z 328.331,A -85,B 0,C 180,E1 27567.358,E2 27567.358} C_VEL
LIN {X 0,Y 609.072,Z 328.316,A -85,B 0,C 180,E1 27564.025,E2 27564.025} C_VEL
LIN {X 0,Y 609.071,Z 328.348,A -85,B 0,C 180,E1 27560.769,E2 27560.769} C_VEL
LIN {X 0,Y 609.062,Z 328.349,A -85,B 0,C 180,E1 27557.385,E2 27557.385} C_VEL
LIN {X 0,Y 609.079,Z 328.365,A -85,B 0,C 180,E1 27554.159,E2 27554.159} C_VEL
LIN {X 0,Y 609.111,Z 328.606,A -85,B 0,C 180,E1 27553.673,E2 27553.673} C_VEL
LIN {X 0,Y 613.159,Z 342.274,A -85,B 0,C 180,E1 27553.077,E2 27553.077} C_VEL
LIN {X 0,Y 613.159,Z 422.069,A -85,B 0,C 180,E1 27550.31,E2 27550.31} C_VEL
LIN {X 0,Y 613.547,Z 503.264,A -85,B 0,C 180,E1 27547.35,E2 27547.35} C_VEL
LIN {X 0,Y 613.565,Z 576.695,A -85,B 0,C 180,E1 27544.58,E2 27544.58} C_VEL
LIN {X 0,Y 613.145,Z 655.395,A -85,B 0,C 180,E1 27541.542,E2 27541.542} C_VEL
LIN {X 0,Y 612.443,Z 733.458,A -85,B 0,C 180,E1 27538.456,E2 27538.456} C_VEL
LIN {X 0,Y 611.643,Z 808.397,A -85,B 0,C 180,E1 27535.452,E2 27535.452} C_VEL
LIN {X 0,Y 611.028,Z 847.122,A -85,B 0,C 180,E1 27533.894,E2 27533.894} C_VEL
LIN {X 0,Y 610.773,Z 851.599,A -85,B 0,C 180,E1 27533.748,E2 27533.748} C_VEL
LIN {X 0,Y 610.245,Z 965.53,A -85,B 0,C 180,E1 27532.347,E2 27532.347} C_VEL
LIN {X 0,Y 610.243,Z 977.859,A -85,B 0,C 180,E1 27532.072,E2 27532.072} C_VEL
LIN {X 0,Y 610.2,Z 989.126,A -85,B 0,C 180,E1 27531.709,E2 27531.709} C_VEL
LIN {X 0,Y 610.096,Z 1001.193,A -85,B 0,C 180,E1 27531.19,E2 27531.19} C_VEL
LIN {X 0,Y 609.898,Z 1014.561,A -85,B 0,C 180,E1 27530.421,E2 27530.421} C_VEL
LIN {X 0,Y 609.713,Z 1024.834,A -85,B 0,C 180,E1 27529.655,E2 27529.655} C_VEL
LIN {X 0,Y 609.531,Z 1032.796,A -85,B 0,C 180,E1 27528.935,E2 27528.935} C_VEL
LIN {X 0,Y 609.339,Z 1040.702,A -85,B 0,C 180,E1 27528.067,E2 27528.067} C_VEL
LIN {X 0,Y 609.172,Z 1047.467,A -85,B 0,C 180,E1 27527.159,E2 27527.159} C_VEL
LIN {X 0,Y 609.003,Z 1054.297,A -85,B 0,C 180,E1 27526.01,E2 27526.01} C_VEL
LIN {X 0,Y 608.85,Z 1060.004,A -85,B 0,C 180,E1 27524.668,E2 27524.668} C_VEL
LIN {X 0,Y 608.768,Z 1063.215,A -85,B 0,C 180,E1 27523.58,E2 27523.58} C_VEL
LIN {X 0,Y 608.721,Z 1065.227,A -85,B 0,C 180,E1 27522.506,E2 27522.506} C_VEL
LIN {X 0,Y 608.69,Z 1066.158,A -85,B 0,C 180,E1 27521.412,E2 27521.412} C_VEL
LIN {X 0,Y 608.681,Z 1065.95,A -85,B 0,C 180,E1 27520.268,E2 27520.268} C_VEL
LIN {X 0,Y 608.699,Z 1064.208,A -85,B 0,C 180,E1 27518.914,E2 27518.914} C_VEL
LIN {X 0,Y 608.758,Z 1060.676,A -85,B 0,C 180,E1 27517.6,E2 27517.6} C_VEL
LIN {X 0,Y 608.833,Z 1056.285,A -85,B 0,C 180,E1 27516.479,E2 27516.479} C_VEL
LIN {X 0,Y 608.946,Z 1051.004,A -85,B 0,C 180,E1 27515.454,E2 27515.454} C_VEL
LIN {X 0,Y 609.106,Z 1044.292,A -85,B 0,C 180,E1 27514.422,E2 27514.422} C_VEL
LIN {X 0,Y 609.346,Z 1034.848,A -85,B 0,C 180,E1 27513.281,E2 27513.281} C_VEL
LIN {X 0,Y 609.572,Z 1024.898,A -85,B 0,C 180,E1 27512.347,E2 27512.347} C_VEL
LIN {X 0,Y 609.758,Z 1015.192,A -85,B 0,C 180,E1 27511.605,E2 27511.605} C_VEL
LIN {X 0,Y 609.955,Z 1005.031,A -85,B 0,C 180,E1 27510.972,E2 27510.972} C_VEL
LIN {X 0,Y 610.148,Z 992.148,A -85,B 0,C 180,E1 27510.336,E2 27510.336} C_VEL
LIN {X 0,Y 610.243,Z 977.673,A -85,B 0,C 180,E1 27509.834,E2 27509.834} C_VEL
LIN {X 0,Y 610.284,Z 965.304,A -85,B 0,C 180,E1 27509.541,E2 27509.541} C_VEL
LIN {X 0,Y 610.278,Z 946.619,A -85,B 0,C 180,E1 27509.279,E2 27509.279} C_VEL
LIN {X 0,Y 610.318,Z 939.106,A -85,B 0,C 180,E1 27509.191,E2 27509.191} C_VEL
LIN {X 0,Y 609.368,Z 931.484,A -85,B 0,C 180,E1 27509.082,E2 27509.082} C_VEL
LIN {X 0,Y 603.35,Z 911.462,A -85,B 0,C 180,E1 27508.723,E2 27508.723} C_VEL
LIN {X 0,Y 602.656,Z 904.915,A -85,B 0,C 180,E1 27508.628,E2 27508.628} C_VEL
LIN {X 0,Y 603.081,Z 847.912,A -85,B 0,C 180,E1 27507.912,E2 27507.912} C_VEL
LIN {X 0,Y 603.921,Z 802.86,A -85,B 0,C 180,E1 27506.047,E2 27506.047} C_VEL
LIN {X 0,Y 605.109,Z 723.157,A -85,B 0,C 180,E1 27502.732,E2 27502.732} C_VEL
LIN {X 0,Y 606.325,Z 645.014,A -85,B 0,C 180,E1 27499.477,E2 27499.477} C_VEL
LIN {X 0,Y 606.634,Z 626.641,A -85,B 0,C 180,E1 27498.706,E2 27498.706} C_VEL
LIN {X 0,Y 607.714,Z 628.394,A -85,B 0,C 180,E1 27498.56,E2 27498.56} C_VEL
LIN {X 0,Y 609.622,Z 628.516,A -85,B 0,C 180,E1 27498.373,E2 27498.373} C_VEL
LIN {X 0,Y 612.465,Z 626.316,A -85,B 0,C 180,E1 27498.155,E2 27498.155} C_VEL
LIN {X 0,Y 616.146,Z 620.858,A -85,B 0,C 180,E1 27497.931,E2 27497.931} C_VEL
LIN {X 0,Y 616.991,Z 620.476,A -85,B 0,C 180,E1 27497.861,E2 27497.861} C_VEL
LIN {X 0,Y 620.562,Z 618.9,A -85,B 0,C 180,E1 27497.568,E2 27497.568} C_VEL
LIN {X 0,Y 624.587,Z 614.977,A -85,B 0,C 180,E1 27497.283,E2 27497.283} C_VEL
LIN {X 0,Y 626.933,Z 611.663,A -85,B 0,C 180,E1 27497.139,E2 27497.139} C_VEL
LIN {X 0,Y 631.566,Z 609.006,A -85,B 0,C 180,E1 27496.785,E2 27496.785} C_VEL
LIN {X 0,Y 636.245,Z 604.226,A -85,B 0,C 180,E1 27496.47,E2 27496.47} C_VEL
LIN {X 0,Y 638.102,Z 601.952,A -85,B 0,C 180,E1 27496.35,E2 27496.35} C_VEL
LIN {X 0,Y 639.365,Z 601.477,A -85,B 0,C 180,E1 27496.253,E2 27496.253} C_VEL
LIN {X 0,Y 637.034,Z 726.363,A -85,B 0,C 180,E1 27494.597,E2 27494.597} C_VEL
LIN {X 0,Y 635.559,Z 794.958,A -85,B 0,C 180,E1 27493.675,E2 27493.675} C_VEL
LIN {X 0,Y 634.584,Z 816.042,A -85,B 0,C 180,E1 27493.311,E2 27493.311} C_VEL
LIN {X 0,Y 633.354,Z 836.635,A -85,B 0,C 180,E1 27492.855,E2 27492.855} C_VEL
LIN {X 0,Y 631.877,Z 857.188,A -85,B 0,C 180,E1 27492.294,E2 27492.294} C_VEL
LIN {X 0,Y 630.164,Z 878.035,A -85,B 0,C 180,E1 27491.609,E2 27491.609} C_VEL
LIN {X 0,Y 628.221,Z 899.113,A -85,B 0,C 180,E1 27490.796,E2 27490.796} C_VEL
LIN {X 0,Y 625.71,Z 924.011,A -85,B 0,C 180,E1 27489.674,E2 27489.674} C_VEL
LIN {X 0,Y 622.872,Z 948.752,A -85,B 0,C 180,E1 27488.349,E2 27488.349} C_VEL
LIN {X 0,Y 620.45,Z 968.778,A -85,B 0,C 180,E1 27487.124,E2 27487.124} C_VEL
LIN {X 0,Y 618.132,Z 987.412,A -85,B 0,C 180,E1 27485.844,E2 27485.844} C_VEL
LIN {X 0,Y 615.739,Z 1006.131,A -85,B 0,C 180,E1 27484.411,E2 27484.411} C_VEL
LIN {X 0,Y 613.074,Z 1027.038,A -85,B 0,C 180,E1 27482.618,E2 27482.618} C_VEL
LIN {X 0,Y 610.344,Z 1048.674,A -85,B 0,C 180,E1 27480.49,E2 27480.49} C_VEL
LIN {X 0,Y 608.217,Z 1065.881,A -85,B 0,C 180,E1 27478.581,E2 27478.581} C_VEL
LIN {X 0,Y 606.379,Z 1081.522,A -85,B 0,C 180,E1 27476.649,E2 27476.649} C_VEL
LIN {X 0,Y 604.605,Z 1098.319,A -85,B 0,C 180,E1 27474.318,E2 27474.318} C_VEL
LIN {X 0,Y 603.175,Z 1112.812,A -85,B 0,C 180,E1 27472.003,E2 27472.003} C_VEL
LIN {X 0,Y 602.221,Z 1123.968,A -85,B 0,C 180,E1 27470.001,E2 27470.001} C_VEL
LIN {X 0,Y 601.473,Z 1133.764,A -85,B 0,C 180,E1 27468.029,E2 27468.029} C_VEL
LIN {X 0,Y 600.924,Z 1142.511,A -85,B 0,C 180,E1 27466.035,E2 27466.035} C_VEL
LIN {X 0,Y 600.493,Z 1150.754,A -85,B 0,C 180,E1 27463.874,E2 27463.874} C_VEL
LIN {X 0,Y 600.201,Z 1158.32,A -85,B 0,C 180,E1 27461.533,E2 27461.533} C_VEL
LIN {X 0,Y 600.014,Z 1165.264,A -85,B 0,C 180,E1 27458.808,E2 27458.808} C_VEL
LIN {X 0,Y 599.945,Z 1169.776,A -85,B 0,C 180,E1 27456.412,E2 27456.412} C_VEL
LIN {X 0,Y 599.918,Z 1172.795,A -85,B 0,C 180,E1 27454.111,E2 27454.111} C_VEL
LIN {X 0,Y 599.91,Z 1174.461,A -85,B 0,C 180,E1 27451.911,E2 27451.911} C_VEL
LIN {X 0,Y 599.893,Z 1174.934,A -85,B 0,C 180,E1 27449.428,E2 27449.428} C_VEL
LIN {X 0,Y 599.913,Z 1173.798,A -85,B 0,C 180,E1 27446.848,E2 27446.848} C_VEL
LIN {X 0,Y 599.93,Z 1170.945,A -85,B 0,C 180,E1 27444.262,E2 27444.262} C_VEL
LIN {X 0,Y 599.984,Z 1167.003,A -85,B 0,C 180,E1 27441.954,E2 27441.954} C_VEL
LIN {X 0,Y 600.092,Z 1161.959,A -85,B 0,C 180,E1 27439.731,E2 27439.731} C_VEL
LIN {X 0,Y 600.287,Z 1155.621,A -85,B 0,C 180,E1 27437.496,E2 27437.496} C_VEL
LIN {X 0,Y 600.641,Z 1147.897,A -85,B 0,C 180,E1 27435.246,E2 27435.246} C_VEL
LIN {X 0,Y 601.273,Z 1137.049,A -85,B 0,C 180,E1 27432.584,E2 27432.584} C_VEL
LIN {X 0,Y 602.067,Z 1126.007,A -85,B 0,C 180,E1 27430.299,E2 27430.299} C_VEL
LIN {X 0,Y 602.909,Z 1115.673,A -85,B 0,C 180,E1 27428.399,E2 27428.399} C_VEL
LIN {X 0,Y 604.001,Z 1104.087,A -85,B 0,C 180,E1 27426.488,E2 27426.488} C_VEL
LIN {X 0,Y 605.316,Z 1091.132,A -85,B 0,C 180,E1 27424.567,E2 27424.567} C_VEL
LIN {X 0,Y 607.061,Z 1075.878,A -85,B 0,C 180,E1 27422.538,E2 27422.538} C_VEL
LIN {X 0,Y 609.486,Z 1055.411,A -85,B 0,C 180,E1 27420.137,E2 27420.137} C_VEL
LIN {X 0,Y 611.793,Z 1037.06,A -85,B 0,C 180,E1 27418.249,E2 27418.249} C_VEL
LIN {X 0,Y 614.22,Z 1018.16,A -85,B 0,C 180,E1 27416.507,E2 27416.507} C_VEL
LIN {X 0,Y 617.102,Z 995.576,A -85,B 0,C 180,E1 27414.661,E2 27414.661} C_VEL
LIN {X 0,Y 619.996,Z 972.365,A -85,B 0,C 180,E1 27413.021,E2 27413.021} C_VEL
LIN {X 0,Y 622.377,Z 952.725,A -85,B 0,C 180,E1 27411.793,E2 27411.793} C_VEL
LIN {X 0,Y 624.6,Z 933.416,A -85,B 0,C 180,E1 27410.72,E2 27410.72} C_VEL
LIN {X 0,Y 626.849,Z 912.592,A -85,B 0,C 180,E1 27409.7,E2 27409.7} C_VEL
LIN {X 0,Y 629.453,Z 886.669,A -85,B 0,C 180,E1 27408.61,E2 27408.61} C_VEL
LIN {X 0,Y 631.654,Z 860.202,A -85,B 0,C 180,E1 27407.707,E2 27407.707} C_VEL
LIN {X 0,Y 633.233,Z 838.565,A -85,B 0,C 180,E1 27407.103,E2 27407.103} C_VEL
LIN {X 0,Y 634.51,Z 817.479,A -85,B 0,C 180,E1 27406.627,E2 27406.627} C_VEL
LIN {X 0,Y 635.508,Z 796.302,A -85,B 0,C 180,E1 27406.256,E2 27406.256} C_VEL
LIN {X 0,Y 636.948,Z 732.304,A -85,B 0,C 180,E1 27405.389,E2 27405.389} C_VEL
LIN {X 0,Y 639.314,Z 603.138,A -85,B 0,C 180,E1 27403.681,E2 27403.681} C_VEL
LIN {X 0,Y 645.279,Z 388.437,A -85,B 0,C 180,E1 27400.622,E2 27400.622} C_VEL
LIN {X 0,Y 640.066,Z 381.224,A -85,B 0,C 180,E1 27399.945,E2 27399.945} C_VEL
LIN {X 0,Y 625.314,Z 367.112,A -85,B 0,C 180,E1 27398.027,E2 27398.027} C_VEL
LIN {X 0,Y 619.859,Z 361.823,A -85,B 0,C 180,E1 27397.252,E2 27397.252} C_VEL
LIN {X 0,Y 616.275,Z 355.612,A -85,B 0,C 180,E1 27395.467,E2 27395.467} C_VEL
LIN {X 0,Y 614.153,Z 351.702,A -85,B 0,C 180,E1 27394.286,E2 27394.286} C_VEL
LIN {X 0,Y 611.184,Z 346.59,A -85,B 0,C 180,E1 27392.564,E2 27392.564} C_VEL
LIN {X 0,Y 610.329,Z 345.243,A -85,B 0,C 180,E1 27392.06,E2 27392.06} C_VEL
LIN {X 0,Y 608.208,Z 341.733,A -85,B 0,C 180,E1 27390.709,E2 27390.709} C_VEL
LIN {X 0,Y 607.657,Z 340.322,A -85,B 0,C 180,E1 27390.233,E2 27390.233} C_VEL
LIN {X 0,Y 605.072,Z 336.751,A -85,B 0,C 180,E1 27388.527,E2 27388.527} C_VEL
LIN {X 0,Y 604.401,Z 334.853,A -85,B 0,C 180,E1 27387.809,E2 27387.809} C_VEL
LIN {X 0,Y 601.704,Z 331.496,A -85,B 0,C 180,E1 27385.758,E2 27385.758} C_VEL
LIN {X 0,Y 601.11,Z 329.307,A -85,B 0,C 180,E1 27384.744,E2 27384.744} C_VEL
LIN {X 0,Y 601.138,Z 329.325,A -85,B 0,C 180,E1 27381.568,E2 27381.568} C_VEL
LIN {X 0,Y 601.133,Z 329.352,A -85,B 0,C 180,E1 27378.122,E2 27378.122} C_VEL
LIN {X 0,Y 601.141,Z 329.309,A -85,B 0,C 180,E1 27374.743,E2 27374.743} C_VEL
LIN {X 0,Y 601.105,Z 329.312,A -85,B 0,C 180,E1 27371.612,E2 27371.612} C_VEL
LIN {X 0,Y 601.118,Z 329.356,A -85,B 0,C 180,E1 27368.417,E2 27368.417} C_VEL
LIN {X 0,Y 601.127,Z 329.312,A -85,B 0,C 180,E1 27365.249,E2 27365.249} C_VEL
LIN {X 0,Y 601.145,Z 329.59,A -85,B 0,C 180,E1 27363.337,E2 27363.337} C_VEL
LIN {X 0,Y 602.906,Z 333.438,A -85,B 0,C 180,E1 27361.425,E2 27361.425} C_VEL
LIN {X 0,Y 604.645,Z 335.173,A -85,B 0,C 180,E1 27360.284,E2 27360.284} C_VEL
LIN {X 0,Y 606.217,Z 338.828,A -85,B 0,C 180,E1 27358.866,E2 27358.866} C_VEL
LIN {X 0,Y 608.013,Z 340.863,A -85,B 0,C 180,E1 27357.832,E2 27357.832} C_VEL
LIN {X 0,Y 609.841,Z 344.632,A -85,B 0,C 180,E1 27356.522,E2 27356.522} C_VEL
LIN {X 0,Y 611.251,Z 346.431,A -85,B 0,C 180,E1 27355.779,E2 27355.779} C_VEL
LIN {X 0,Y 613.219,Z 350.218,A -85,B 0,C 180,E1 27354.573,E2 27354.573} C_VEL
LIN {X 0,Y 614.361,Z 351.739,A -85,B 0,C 180,E1 27354.021,E2 27354.021} C_VEL
LIN {X 0,Y 616.337,Z 355.543,A -85,B 0,C 180,E1 27352.918,E2 27352.918} C_VEL
LIN {X 0,Y 617.455,Z 357.374,A -85,B 0,C 180,E1 27352.369,E2 27352.369} C_VEL
LIN {X 0,Y 620.444,Z 362.686,A -85,B 0,C 180,E1 27350.913,E2 27350.913} C_VEL
LIN {X 0,Y 623.374,Z 368.045,A -85,B 0,C 180,E1 27349.557,E2 27349.557} C_VEL
LIN {X 0,Y 626.025,Z 372.963,A -85,B 0,C 180,E1 27348.39,E2 27348.39} C_VEL
LIN {X 0,Y 630.577,Z 381.353,A -85,B 0,C 180,E1 27346.521,E2 27346.521} C_VEL
LIN {X 0,Y 637.413,Z 394.683,A -85,B 0,C 180,E1 27343.88,E2 27343.88} C_VEL
LIN {X 0,Y 644.087,Z 408.521,A -85,B 0,C 180,E1 27341.455,E2 27341.455} C_VEL
LIN {X 0,Y 640.482,Z 441.239,A -85,B 0,C 180,E1 27338.745,E2 27338.745} C_VEL
LIN {X 0,Y 636.793,Z 477.124,A -85,B 0,C 180,E1 27335.905,E2 27335.905} C_VEL
LIN {X 0,Y 633.024,Z 516.242,A -85,B 0,C 180,E1 27332.941,E2 27332.941} C_VEL
LIN {X 0,Y 629.426,Z 556.291,A -85,B 0,C 180,E1 27330.021,E2 27330.021} C_VEL
LIN {X 0,Y 628.409,Z 576.516,A -85,B 0,C 180,E1 27328.52,E2 27328.52} C_VEL
LIN {X 0,Y 629.355,Z 591.943,A -85,B 0,C 180,E1 27327.25,E2 27327.25} C_VEL
LIN {X 0,Y 632.084,Z 605.775,A -85,B 0,C 180,E1 27325.984,E2 27325.984} C_VEL
LIN {X 0,Y 636.678,Z 618.427,A -85,B 0,C 180,E1 27324.694,E2 27324.694} C_VEL
LIN {X 0,Y 642.932,Z 629.438,A -85,B 0,C 180,E1 27323.441,E2 27323.441} C_VEL
LIN {X 0,Y 650.415,Z 638.587,A -85,B 0,C 180,E1 27322.276,E2 27322.276} C_VEL
LIN {X 0,Y 659.527,Z 646.629,A -85,B 0,C 180,E1 27321.123,E2 27321.123} C_VEL
LIN {X 0,Y 670.33,Z 653.44,A -85,B 0,C 180,E1 27319.992,E2 27319.992} C_VEL
LIN {X 0,Y 682.905,Z 658.837,A -85,B 0,C 180,E1 27318.897,E2 27318.897} C_VEL
LIN {X 0,Y 687.855,Z 660.268,A -85,B 0,C 180,E1 27318.482,E2 27318.482} C_VEL
LIN {X 0,Y 691.808,Z 660.47,A -85,B 0,C 180,E1 27317.995,E2 27317.995} C_VEL
LIN {X 0,Y 694.238,Z 659.551,A -85,B 0,C 180,E1 27317.508,E2 27317.508} C_VEL
LIN {X 0,Y 695.349,Z 657.761,A -85,B 0,C 180,E1 27317.031,E2 27317.031} C_VEL
LIN {X 0,Y 695.137,Z 654.871,A -85,B 0,C 180,E1 27316.529,E2 27316.529} C_VEL
LIN {X 0,Y 693.926,Z 652.421,A -85,B 0,C 180,E1 27316.183,E2 27316.183} C_VEL
LIN {X 0,Y 689.376,Z 668.86,A -85,B 0,C 180,E1 27316.194,E2 27316.194} C_VEL
LIN {X 0,Y 682.821,Z 685.308,A -85,B 0,C 180,E1 27316.211,E2 27316.211} C_VEL
LIN {X 0,Y 673.979,Z 702.368,A -85,B 0,C 180,E1 27316.176,E2 27316.176} C_VEL
LIN {X 0,Y 666.67,Z 714.853,A -85,B 0,C 180,E1 27316.045,E2 27316.045} C_VEL
LIN {X 0,Y 660.524,Z 725.942,A -85,B 0,C 180,E1 27315.787,E2 27315.787} C_VEL
LIN {X 0,Y 653.289,Z 736.835,A -85,B 0,C 180,E1 27315.616,E2 27315.616} C_VEL
LIN {X 0,Y 647.51,Z 746.983,A -85,B 0,C 180,E1 27315.323,E2 27315.323} C_VEL
LIN {X 0,Y 644.329,Z 753.269,A -85,B 0,C 180,E1 27315.103,E2 27315.103} C_VEL
LIN {X 0,Y 640.04,Z 761.903,A -85,B 0,C 180,E1 27314.792,E2 27314.792} C_VEL
LIN {X 0,Y 636.916,Z 769.861,A -85,B 0,C 180,E1 27314.478,E2 27314.478} C_VEL
LIN {X 0,Y 635.368,Z 830.601,A -85,B 0,C 180,E1 27313.636,E2 27313.636} C_VEL
LIN {X 0,Y 633.944,Z 857.937,A -85,B 0,C 180,E1 27313.109,E2 27313.109} C_VEL
LIN {X 0,Y 632.196,Z 883.768,A -85,B 0,C 180,E1 27312.444,E2 27312.444} C_VEL
LIN {X 0,Y 630.098,Z 909.443,A -85,B 0,C 180,E1 27311.612,E2 27311.612} C_VEL
LIN {X 0,Y 627.802,Z 933.804,A -85,B 0,C 180,E1 27310.646,E2 27310.646} C_VEL
LIN {X 0,Y 625.272,Z 957.792,A -85,B 0,C 180,E1 27309.526,E2 27309.526} C_VEL
LIN {X 0,Y 622.702,Z 980.49,A -85,B 0,C 180,E1 27308.3,E2 27308.3} C_VEL
LIN {X 0,Y 619.702,Z 1004.986,A -85,B 0,C 180,E1 27306.768,E2 27306.768} C_VEL
LIN {X 0,Y 616.745,Z 1028.417,A -85,B 0,C 180,E1 27305.073,E2 27305.073} C_VEL
LIN {X 0,Y 614.078,Z 1049.273,A -85,B 0,C 180,E1 27303.352,E2 27303.352} C_VEL
LIN {X 0,Y 611.378,Z 1070.44,A -85,B 0,C 180,E1 27301.381,E2 27301.381} C_VEL
LIN {X 0,Y 609.025,Z 1089.183,A -85,B 0,C 180,E1 27299.398,E2 27299.398} C_VEL
LIN {X 0,Y 606.801,Z 1108.003,A -85,B 0,C 180,E1 27297.149,E2 27297.149} C_VEL
LIN {X 0,Y 605.119,Z 1123.14,A -85,B 0,C 180,E1 27295.108,E2 27295.108} C_VEL
LIN {X 0,Y 603.521,Z 1139.223,A -85,B 0,C 180,E1 27292.658,E2 27292.658} C_VEL
LIN {X 0,Y 602.318,Z 1152.753,A -85,B 0,C 180,E1 27290.291,E2 27290.291} C_VEL
LIN {X 0,Y 601.467,Z 1164.106,A -85,B 0,C 180,E1 27288.01,E2 27288.01} C_VEL
LIN {X 0,Y 600.781,Z 1174.927,A -85,B 0,C 180,E1 27285.497,E2 27285.497} C_VEL
LIN {X 0,Y 600.353,Z 1184.281,A -85,B 0,C 180,E1 27282.894,E2 27282.894} C_VEL
LIN {X 0,Y 600.1,Z 1191.662,A -85,B 0,C 180,E1 27280.366,E2 27280.366} C_VEL
LIN {X 0,Y 599.979,Z 1197.331,A -85,B 0,C 180,E1 27277.853,E2 27277.853} C_VEL
LIN {X 0,Y 599.927,Z 1201.414,A -85,B 0,C 180,E1 27275.354,E2 27275.354} C_VEL
LIN {X 0,Y 599.915,Z 1203.98,A -85,B 0,C 180,E1 27272.865,E2 27272.865} C_VEL
LIN {X 0,Y 599.892,Z 1204.916,A -85,B 0,C 180,E1 27270.476,E2 27270.476} C_VEL
LIN {X 0,Y 599.911,Z 1204.415,A -85,B 0,C 180,E1 27267.897,E2 27267.897} C_VEL
LIN {X 0,Y 599.916,Z 1202.393,A -85,B 0,C 180,E1 27265.41,E2 27265.41} C_VEL
LIN {X 0,Y 599.955,Z 1198.773,A -85,B 0,C 180,E1 27262.915,E2 27262.915} C_VEL
LIN {X 0,Y 600.051,Z 1193.556,A -85,B 0,C 180,E1 27260.407,E2 27260.407} C_VEL
LIN {X 0,Y 600.244,Z 1186.733,A -85,B 0,C 180,E1 27257.883,E2 27257.883} C_VEL
LIN {X 0,Y 600.592,Z 1178.838,A -85,B 0,C 180,E1 27255.538,E2 27255.538} C_VEL
LIN {X 0,Y 601.133,Z 1169.014,A -85,B 0,C 180,E1 27253.076,E2 27253.076} C_VEL
LIN {X 0,Y 602.001,Z 1156.842,A -85,B 0,C 180,E1 27250.496,E2 27250.496} C_VEL
LIN {X 0,Y 603.055,Z 1144.316,A -85,B 0,C 180,E1 27248.197,E2 27248.197} C_VEL
LIN {X 0,Y 604.426,Z 1129.901,A -85,B 0,C 180,E1 27245.882,E2 27245.882} C_VEL
LIN {X 0,Y 606.187,Z 1113.396,A -85,B 0,C 180,E1 27243.553,E2 27243.553} C_VEL
LIN {X 0,Y 607.952,Z 1097.996,A -85,B 0,C 180,E1 27241.619,E2 27241.619} C_VEL
LIN {X 0,Y 610.364,Z 1078.514,A -85,B 0,C 180,E1 27239.445,E2 27239.445} C_VEL
LIN {X 0,Y 612.827,Z 1058.966,A -85,B 0,C 180,E1 27237.516,E2 27237.516} C_VEL
LIN {X 0,Y 615.685,Z 1036.7,A -85,B 0,C 180,E1 27235.586,E2 27235.586} C_VEL
LIN {X 0,Y 618.604,Z 1013.737,A -85,B 0,C 180,E1 27233.844,E2 27233.844} C_VEL
LIN {X 0,Y 621.276,Z 992.332,A -85,B 0,C 180,E1 27232.412,E2 27232.412} C_VEL
LIN {X 0,Y 624.274,Z 966.719,A -85,B 0,C 180,E1 27230.93,E2 27230.93} C_VEL
LIN {X 0,Y 626.965,Z 941.831,A -85,B 0,C 180,E1 27229.706,E2 27229.706} C_VEL
LIN {X 0,Y 629.407,Z 916.786,A -85,B 0,C 180,E1 27228.664,E2 27228.664} C_VEL
LIN {X 0,Y 631.702,Z 889.846,A -85,B 0,C 180,E1 27227.738,E2 27227.738} C_VEL
LIN {X 0,Y 633.582,Z 863.952,A -85,B 0,C 180,E1 27227.029,E2 27227.029} C_VEL
LIN {X 0,Y 635.068,Z 837.715,A -85,B 0,C 180,E1 27226.481,E2 27226.481} C_VEL
LIN {X 0,Y 636.133,Z 806.014,A -85,B 0,C 180,E1 27226.011,E2 27226.011} C_VEL
LIN {X 0,Y 637.346,Z 759.125,A -85,B 0,C 180,E1 27225.36,E2 27225.36} C_VEL
LIN {X 0,Y 642.196,Z 695.926,A -85,B 0,C 180,E1 27224.305,E2 27224.305} C_VEL
LIN {X 0,Y 645.034,Z 660.123,A -85,B 0,C 180,E1 27223.713,E2 27223.713} C_VEL
LIN {X 0,Y 646.454,Z 644.02,A -85,B 0,C 180,E1 27223.46,E2 27223.46} C_VEL
LIN {X 0,Y 649.239,Z 611.444,A -85,B 0,C 180,E1 27222.939,E2 27222.939} C_VEL
LIN {X 0,Y 651.134,Z 593.229,A -85,B 0,C 180,E1 27222.677,E2 27222.677} C_VEL
LIN {X 0,Y 653.135,Z 567.121,A -85,B 0,C 180,E1 27222.239,E2 27222.239} C_VEL
LIN {X 0,Y 656.773,Z 535.105,A -85,B 0,C 180,E1 27221.808,E2 27221.808} C_VEL
LIN {X 0,Y 658.291,Z 513.142,A -85,B 0,C 180,E1 27221.424,E2 27221.424} C_VEL
LIN {X 0,Y 662.17,Z 480.827,A -85,B 0,C 180,E1 27221.01,E2 27221.01} C_VEL
LIN {X 0,Y 663.23,Z 472.093,A -85,B 0,C 180,E1 27220.9,E2 27220.9} C_VEL
LIN {X 0,Y 664.298,Z 453.699,A -85,B 0,C 180,E1 27220.559,E2 27220.559} C_VEL
LIN {X 0,Y 667.705,Z 424.621,A -85,B 0,C 180,E1 27220.18,E2 27220.18} C_VEL
LIN {X 0,Y 668.891,Z 415.589,A -85,B 0,C 180,E1 27220.075,E2 27220.075} C_VEL
LIN {X 0,Y 660.577,Z 409.117,A -85,B 0,C 180,E1 27219.111,E2 27219.111} C_VEL
LIN {X 0,Y 650.738,Z 398.662,A -85,B 0,C 180,E1 27217.841,E2 27217.841} C_VEL
LIN {X 0,Y 634.827,Z 375.572,A -85,B 0,C 180,E1 27215.452,E2 27215.452} C_VEL
LIN {X 0,Y 624.993,Z 361.91,A -85,B 0,C 180,E1 27213.862,E2 27213.862} C_VEL
LIN {X 0,Y 620.769,Z 356.286,A -85,B 0,C 180,E1 27213.151,E2 27213.151} C_VEL
LIN {X 0,Y 617.345,Z 351.679,A -85,B 0,C 180,E1 27212.557,E2 27212.557} C_VEL
LIN {X 0,Y 613.401,Z 346.379,A -85,B 0,C 180,E1 27211.853,E2 27211.853} C_VEL
LIN {X 0,Y 610.322,Z 342.254,A -85,B 0,C 180,E1 27211.288,E2 27211.288} C_VEL
LIN {X 0,Y 609.182,Z 340.82,A -85,B 0,C 180,E1 27211.079,E2 27211.079} C_VEL
LIN {X 0,Y 606.345,Z 337.373,A -85,B 0,C 180,E1 27210.552,E2 27210.552} C_VEL
LIN {X 0,Y 605.202,Z 335.307,A -85,B 0,C 180,E1 27210.314,E2 27210.314} C_VEL
LIN {X 0,Y 602.421,Z 332.784,A -85,B 0,C 180,E1 27209.809,E2 27209.809} C_VEL
LIN {X 0,Y 601.189,Z 329.864,A -85,B 0,C 180,E1 27209.52,E2 27209.52} C_VEL
LIN {X 0,Y 601.103,Z 329.327,A -85,B 0,C 180,E1 27209.475,E2 27209.475} C_VEL
LIN {X 0,Y 601.121,Z 329.287,A -85,B 0,C 180,E1 27206.367,E2 27206.367} C_VEL
LIN {X 0,Y 601.114,Z 329.338,A -85,B 0,C 180,E1 27203.218,E2 27203.218} C_VEL
LIN {X 0,Y 601.14,Z 329.339,A -85,B 0,C 180,E1 27199.937,E2 27199.937} C_VEL
LIN {X 0,Y 601.119,Z 329.337,A -85,B 0,C 180,E1 27196.724,E2 27196.724} C_VEL
LIN {X 0,Y 601.152,Z 329.427,A -85,B 0,C 180,E1 27193.916,E2 27193.916} C_VEL
LIN {X 0,Y 605.571,Z 344.791,A -85,B 0,C 180,E1 27193.244,E2 27193.244} C_VEL
LIN {X 0,Y 605.528,Z 423.829,A -85,B 0,C 180,E1 27190.489,E2 27190.489} C_VEL
LIN {X 0,Y 605.903,Z 504.587,A -85,B 0,C 180,E1 27187.539,E2 27187.539} C_VEL
LIN {X 0,Y 605.898,Z 578.792,A -85,B 0,C 180,E1 27184.733,E2 27184.733} C_VEL
LIN {X 0,Y 605.508,Z 643.046,A -85,B 0,C 180,E1 27182.224,E2 27182.224} C_VEL
LIN {X 0,Y 604.893,Z 717.993,A -85,B 0,C 180,E1 27179.29,E2 27179.29} C_VEL
LIN {X 0,Y 604.05,Z 796.029,A -85,B 0,C 180,E1 27176.156,E2 27176.156} C_VEL
LIN {X 0,Y 603.259,Z 847.575,A -85,B 0,C 180,E1 27174.07,E2 27174.07} C_VEL
LIN {X 0,Y 602.95,Z 852.784,A -85,B 0,C 180,E1 27173.896,E2 27173.896} C_VEL
LIN {X 0,Y 602.391,Z 966.678,A -85,B 0,C 180,E1 27172.471,E2 27172.471} C_VEL
LIN {X 0,Y 602.396,Z 979.052,A -85,B 0,C 180,E1 27172.192,E2 27172.192} C_VEL
LIN {X 0,Y 602.357,Z 989.899,A -85,B 0,C 180,E1 27171.841,E2 27171.841} C_VEL
LIN {X 0,Y 602.257,Z 1001.146,A -85,B 0,C 180,E1 27171.358,E2 27171.358} C_VEL
LIN {X 0,Y 602.077,Z 1014.152,A -85,B 0,C 180,E1 27170.633,E2 27170.633} C_VEL
LIN {X 0,Y 601.869,Z 1025.287,A -85,B 0,C 180,E1 27169.809,E2 27169.809} C_VEL
LIN {X 0,Y 601.653,Z 1034.328,A -85,B 0,C 180,E1 27168.982,E2 27168.982} C_VEL
LIN {X 0,Y 601.473,Z 1041.383,A -85,B 0,C 180,E1 27168.201,E2 27168.201} C_VEL
LIN {X 0,Y 601.299,Z 1047.973,A -85,B 0,C 180,E1 27167.32,E2 27167.32} C_VEL
LIN {X 0,Y 601.135,Z 1053.927,A -85,B 0,C 180,E1 27166.338,E2 27166.338} C_VEL
LIN {X 0,Y 600.99,Z 1059.489,A -85,B 0,C 180,E1 27165.158,E2 27165.158} C_VEL
LIN {X 0,Y 600.865,Z 1063.98,A -85,B 0,C 180,E1 27163.766,E2 27163.766} C_VEL
LIN {X 0,Y 600.802,Z 1066.286,A -85,B 0,C 180,E1 27162.568,E2 27162.568} C_VEL
LIN {X 0,Y 600.769,Z 1067.253,A -85,B 0,C 180,E1 27161.464,E2 27161.464} C_VEL
LIN {X 0,Y 600.757,Z 1067.111,A -85,B 0,C 180,E1 27160.354,E2 27160.354} C_VEL
LIN {X 0,Y 600.765,Z 1065.689,A -85,B 0,C 180,E1 27159.134,E2 27159.134} C_VEL
LIN {X 0,Y 600.836,Z 1062.239,A -85,B 0,C 180,E1 27157.702,E2 27157.702} C_VEL
LIN {X 0,Y 600.922,Z 1057.514,A -85,B 0,C 180,E1 27156.463,E2 27156.463} C_VEL
LIN {X 0,Y 601.04,Z 1052.256,A -85,B 0,C 180,E1 27155.424,E2 27155.424} C_VEL
LIN {X 0,Y 601.216,Z 1045.329,A -85,B 0,C 180,E1 27154.344,E2 27154.344} C_VEL
LIN {X 0,Y 601.482,Z 1035.126,A -85,B 0,C 180,E1 27153.117,E2 27153.117} C_VEL
LIN {X 0,Y 601.713,Z 1025.56,A -85,B 0,C 180,E1 27152.217,E2 27152.217} C_VEL
LIN {X 0,Y 601.903,Z 1016.202,A -85,B 0,C 180,E1 27151.497,E2 27151.497} C_VEL
LIN {X 0,Y 602.114,Z 1005.58,A -85,B 0,C 180,E1 27150.83,E2 27150.83} C_VEL
LIN {X 0,Y 602.314,Z 991.534,A -85,B 0,C 180,E1 27150.149,E2 27150.149} C_VEL
LIN {X 0,Y 602.401,Z 977.961,A -85,B 0,C 180,E1 27149.686,E2 27149.686} C_VEL
LIN {X 0,Y 602.438,Z 965.749,A -85,B 0,C 180,E1 27149.399,E2 27149.399} C_VEL
LIN {X 0,Y 602.446,Z 943.85,A -85,B 0,C 180,E1 27149.099,E2 27149.099} C_VEL
LIN {X 0,Y 602.656,Z 904.915,A -85,B 0,C 180,E1 27148.628,E2 27148.628} C_VEL
LIN {X 0,Y 601.73,Z 897.296,A -85,B 0,C 180,E1 27148.514,E2 27148.514} C_VEL
LIN {X 0,Y 595.758,Z 877.288,A -85,B 0,C 180,E1 27148.137,E2 27148.137} C_VEL
LIN {X 0,Y 595.087,Z 870.743,A -85,B 0,C 180,E1 27148.038,E2 27148.038} C_VEL
LIN {X 0,Y 595.291,Z 848.57,A -85,B 0,C 180,E1 27147.743,E2 27147.743} C_VEL
LIN {X 0,Y 596.065,Z 811.353,A -85,B 0,C 180,E1 27146.193,E2 27146.193} C_VEL
LIN {X 0,Y 597.307,Z 730.682,A -85,B 0,C 180,E1 27142.82,E2 27142.82} C_VEL
LIN {X 0,Y 598.532,Z 654.398,A -85,B 0,C 180,E1 27139.622,E2 27139.622} C_VEL
LIN {X 0,Y 598.82,Z 643.511,A -85,B 0,C 180,E1 27139.14,E2 27139.14} C_VEL
LIN {X 0,Y 599.783,Z 645.01,A -85,B 0,C 180,E1 27139.004,E2 27139.004} C_VEL
LIN {X 0,Y 601.46,Z 645.131,A -85,B 0,C 180,E1 27138.827,E2 27138.827} C_VEL
LIN {X 0,Y 604.097,Z 643.067,A -85,B 0,C 180,E1 27138.605,E2 27138.605} C_VEL
LIN {X 0,Y 607.771,Z 637.677,A -85,B 0,C 180,E1 27138.36,E2 27138.36} C_VEL
LIN {X 0,Y 608.335,Z 636.632,A -85,B 0,C 180,E1 27138.328,E2 27138.328} C_VEL
LIN {X 0,Y 612.219,Z 635.202,A -85,B 0,C 180,E1 27138.005,E2 27138.005} C_VEL
LIN {X 0,Y 616.094,Z 631.751,A -85,B 0,C 180,E1 27137.723,E2 27137.723} C_VEL
LIN {X 0,Y 619.087,Z 627.734,A -85,B 0,C 180,E1 27137.537,E2 27137.537} C_VEL
LIN {X 0,Y 623.727,Z 625.058,A -85,B 0,C 180,E1 27137.179,E2 27137.179} C_VEL
LIN {X 0,Y 628.556,Z 620.134,A -85,B 0,C 180,E1 27136.856,E2 27136.856} C_VEL
LIN {X 0,Y 630.324,Z 618.177,A -85,B 0,C 180,E1 27136.742,E2 27136.742} C_VEL
LIN {X 0,Y 633.083,Z 616.666,A -85,B 0,C 180,E1 27136.533,E2 27136.533} C_VEL
LIN {X 0,Y 630.532,Z 734.014,A -85,B 0,C 180,E1 27134.937,E2 27134.937} C_VEL
LIN {X 0,Y 629.147,Z 803.444,A -85,B 0,C 180,E1 27134.017,E2 27134.017} C_VEL
LIN {X 0,Y 627.817,Z 831.132,A -85,B 0,C 180,E1 27133.486,E2 27133.486} C_VEL
LIN {X 0,Y 626.238,Z 853.281,A -85,B 0,C 180,E1 27132.909,E2 27132.909} C_VEL
LIN {X 0,Y 624.436,Z 874.453,A -85,B 0,C 180,E1 27132.233,E2 27132.233} C_VEL
LIN {X 0,Y 622.549,Z 894.142,A -85,B 0,C 180,E1 27131.493,E2 27131.493} C_VEL
LIN {X 0,Y 620.414,Z 914.36,A -85,B 0,C 180,E1 27130.616,E2 27130.616} C_VEL
LIN {X 0,Y 618.22,Z 933.676,A -85,B 0,C 180,E1 27129.658,E2 27129.658} C_VEL
LIN {X 0,Y 615.967,Z 952.221,A -85,B 0,C 180,E1 27128.621,E2 27128.621} C_VEL
LIN {X 0,Y 613.638,Z 970.43,A -85,B 0,C 180,E1 27127.482,E2 27127.482} C_VEL
LIN {X 0,Y 611.214,Z 988.821,A -85,B 0,C 180,E1 27126.198,E2 27126.198} C_VEL
LIN {X 0,Y 608.525,Z 1008.683,A -85,B 0,C 180,E1 27124.648,E2 27124.648} C_VEL
LIN {X 0,Y 605.409,Z 1031.61,A -85,B 0,C 180,E1 27122.614,E2 27122.614} C_VEL
LIN {X 0,Y 602.82,Z 1050.903,A -85,B 0,C 180,E1 27120.655,E2 27120.655} C_VEL
LIN {X 0,Y 600.747,Z 1066.755,A -85,B 0,C 180,E1 27118.861,E2 27118.861} C_VEL
LIN {X 0,Y 598.705,Z 1083.094,A -85,B 0,C 180,E1 27116.804,E2 27116.804} C_VEL
LIN {X 0,Y 596.668,Z 1100.916,A -85,B 0,C 180,E1 27114.241,E2 27114.241} C_VEL
LIN {X 0,Y 595.387,Z 1113.398,A -85,B 0,C 180,E1 27112.202,E2 27112.202} C_VEL
LIN {X 0,Y 594.41,Z 1123.971,A -85,B 0,C 180,E1 27110.276,E2 27110.276} C_VEL
LIN {X 0,Y 593.642,Z 1133.381,A -85,B 0,C 180,E1 27108.36,E2 27108.36} C_VEL
LIN {X 0,Y 593.041,Z 1142.105,A -85,B 0,C 180,E1 27106.355,E2 27106.355} C_VEL
LIN {X 0,Y 592.573,Z 1150.049,A -85,B 0,C 180,E1 27104.263,E2 27104.263} C_VEL
LIN {X 0,Y 592.247,Z 1157.436,A -85,B 0,C 180,E1 27101.986,E2 27101.986} C_VEL
LIN {X 0,Y 592.046,Z 1164.384,A -85,B 0,C 180,E1 27099.332,E2 27099.332} C_VEL
LIN {X 0,Y 591.945,Z 1169.517,A -85,B 0,C 180,E1 27096.67,E2 27096.67} C_VEL
LIN {X 0,Y 591.916,Z 1172.598,A -85,B 0,C 180,E1 27094.361,E2 27094.361} C_VEL
LIN {X 0,Y 591.91,Z 1174.361,A -85,B 0,C 180,E1 27092.131,E2 27092.131} C_VEL
